PROGRAM prgObjectCode
  VAR
    asPatternName : ARRAY[0..c_uiMaxIndPattern] OF STRING := ['1000L6S4A', '1000L6S5A', '1000L7S2A', '1000L9S0A', '800L2S6A', '800L4S3A', '800L5S2A', '800L6S0A', '800L6S1A'];  (* palletizing options *)
    iTMPMaxIndShowPattern : INT;
    iMaxIndPattern : INT;
    iMaxIndShowPattern : INT;
    iMaxIndLayer : INT;
    iTMPMaxIndShowLayer : INT;
    iMaxIndShowLayer : INT;
    iMaxIndTool : INT;
    iTMPMaxIndShowTool : INT;
    iMaxIndShowTool : INT;
    asToolName : ARRAY[0..c_uiMaxIndTool] OF STRING;
  END_VAR
  VAR CONSTANT
    c_uiMaxIndPattern : UINT := 19;
    c_uiMaxIndTool : UINT := 4;
  END_VAR
  VAR
    asLayerName : ARRAY[0..c_uiMaxIndLayers] OF STRING := ['layer0', 'layer1', 'layer2', 'layer3', 'layer4', 'layer5'];  (* palletizing options *)
  END_VAR
  VAR CONSTANT
    c_uiMaxIndLayers : UINT := 5;
  END_VAR
  VAR
    sDesiredObjectCode01 : STRING;
    sDesiredObjectCode02 : STRING;
    sCurrentObjectCode01 : STRING;
    sCurrentObjectCode02 : STRING;
    xInit : BOOL := TRUE;
    asBoxName : ARRAY[0..c_uiMaxIndBoxTypes] OF STRING := ['SMALL_BOX', 'BIG_BOX'];
    aiDefaultIndex : ARRAY[0..c_uiMaxIndBoxTypes] OF INT := [0, 0];
    iMaxInd : INT;
    iInd : INT;
    iTMPMaxIndShow : INT;
    iMaxIndShow : INT;
  END_VAR
  VAR CONSTANT
    c_uiNumBoxTypes : UINT := 2;
    c_uiMaxIndBoxTypes : UINT := (c_uiNumBoxTypes - 1);
  END_VAR

                    iMaxInd := TO_INT(XSIZEOF(asBoxName)/XSIZEOF(asBoxName[0])) - 1;
(*------------------------------------*)
// find max ind to show
iTMPMaxIndShow := -1;
FOR iInd := 0 TO iMaxInd DO
	IF asBoxName[iInd] <> '' THEN
		iTMPMaxIndShow := iInd;
	END_IF
END_FOR
IF iTMPMaxIndShow >= 0 THEN
	iMaxIndShow := iTMPMaxIndShow;
END_IF
(*------------------------------------*)
// find max ind to show
IF xInit THEN
	xInit := FALSE;
	FOR iInd := 0 TO iMaxInd DO
		CASE iInd OF 
			0:
				METH_SetObjectCode01(sValue := asBoxName[aiDefaultIndex[iInd]]);
			1:
				METH_SetObjectCode02(sValue := asBoxName[aiDefaultIndex[iInd]]);
		END_CASE
	END_FOR
	
END_IF

(*------------------------------------*)
// PATTERN find max ind to show
iMaxIndPattern := TO_INT(XSIZEOF(asPatternName)/XSIZEOF(asPatternName[0])) - 1;
iTMPMaxIndShowPattern := -1;
FOR iInd := 0 TO iMaxIndPattern DO
	IF asPatternName[iInd] <> '' THEN
		iTMPMaxIndShowPattern := iInd;
	END_IF
END_FOR
IF iTMPMaxIndShowPattern >= 0 THEN
	iMaxIndShowPattern := iTMPMaxIndShowPattern;
END_IF
(*------------------------------------*)
// LAYER find max ind to show
iMaxIndLayer := TO_INT(XSIZEOF(asLayerName)/XSIZEOF(asLayerName[0])) - 1;
iTMPMaxIndShowLayer := -1;
FOR iInd := 0 TO iMaxIndLayer DO
	IF asLayerName[iInd] <> '' THEN
		iTMPMaxIndShowLayer := iInd;
	END_IF
END_FOR
IF iTMPMaxIndShowLayer >= 0 THEN
	iMaxIndShowLayer := iTMPMaxIndShowLayer;
END_IF
(*------------------------------------*)
// LAYER find max ind to show
iMaxIndTool := TO_INT(XSIZEOF(asToolName)/XSIZEOF(asToolName[0])) - 1;
iTMPMaxIndShowTool := -1;
FOR iInd := 0 TO iMaxIndTool DO
	IF asToolName[iInd] <> '' THEN
		iTMPMaxIndShowTool := iInd;
	END_IF
END_FOR
IF iTMPMaxIndShowTool >= 0 THEN
	iMaxIndShowTool := iTMPMaxIndShowTool;
END_IF


(*------------------------------------*)
// set ros interface
prgROS.METH_SetObjectName_Left_01(sValue := sCurrentObjectCode01);
prgROS.METH_SetObjectName_Right_01(sValue := sCurrentObjectCode01);
prgROS.METH_SetObjectName_Left_02(sValue := sCurrentObjectCode02);
prgROS.METH_SetObjectName_Right_02(sValue := sCurrentObjectCode02);
// GVL.g_ROSInterface_01.sObjectCode := sCurrentObjectCode01;
// GVL.g_ROSInterface_02.sObjectCode := sCurrentObjectCode02;
                  

METHOD METH_SetObjectCode01
  VAR_INPUT
    sValue : STRING;
  END_VAR
                          sDesiredObjectCode01 := sValue;
METH_SetObjCode01();
                        
END_METHOD

METHOD METH_SetObjectCode02
  VAR_INPUT
    sValue : STRING;
  END_VAR
                          sDesiredObjectCode02 := sValue;
METH_SetObjCode02();

                        
END_METHOD

METHOD METH_SetObjCode02
                          sCurrentObjectCode02 := sDesiredObjectCode02;
                        
END_METHOD

METHOD METH_SetObjCode01
                          sCurrentObjectCode01 := sDesiredObjectCode01;
                        
END_METHOD
END_PROGRAM

PROGRAM prg_Hmi_ObjectCode
  VAR
    xDIS_SetObjCode01 : BOOL;
    xTB_SetObjCode01 : BOOL;
    iIndexObjectCode01 : INT;
    sDesiredObjectCode01 : STRING;
    xDIS_SetObjCode02 : BOOL;
    xTB_SetObjCode02 : BOOL;
    iIndexObjectCode02 : INT;
    sDesiredObjectCode02 : STRING;
    sCurrentObjectCode01 : STRING;
    sCurrentObjectCode02 : STRING;
    sPrevDesiredObjectCode01 : STRING;
    sPrevDesiredObjectCode02 : STRING;
  END_VAR

                    // Object 01
sDesiredObjectCode01 := prgObjectCode.asBoxName[iIndexObjectCode01];
xDIS_SetObjCode01 := sDesiredObjectCode01 = '';
IF sDesiredObjectCode01 <> sPrevDesiredObjectCode01 AND NOT xDIS_SetObjCode01 THEN
	xTB_SetObjCode01 := TRUE;
END_IF
IF xTB_SetObjCode01 THEN
	xTB_SetObjCode01 := FALSE;
	prgObjectCode.METH_SetObjectCode01(sValue := sDesiredObjectCode01);
END_IF
(*------------------------------------*)
// Object 02
sDesiredObjectCode02 := prgObjectCode.asBoxName[iIndexObjectCode02];
xDIS_SetObjCode02 := sDesiredObjectCode02 = '';
IF sDesiredObjectCode02 <> sPrevDesiredObjectCode02 AND NOT xDIS_SetObjCode02 THEN
	xTB_SetObjCode02 := TRUE;
END_IF
IF xTB_SetObjCode02 THEN
	xTB_SetObjCode02 := FALSE;
	prgObjectCode.METH_SetObjectCode02(sValue := sDesiredObjectCode02);
END_IF
(*------------------------------------*)
sCurrentObjectCode01 := prgObjectCode.sCurrentObjectCode01;
sCurrentObjectCode02 := prgObjectCode.sCurrentObjectCode02;


sPrevDesiredObjectCode01 := sDesiredObjectCode01;
sPrevDesiredObjectCode02 := sDesiredObjectCode02;
                  
END_PROGRAM

PROGRAM prgOPCUAIncas
  VAR
    BoxInfo : INCAS_box_info_struct_t;
    sPrevBoxCode : STRING;
    sCurrentBoxCode : STRING;
    xThereIsANewBox : BOOL;
    INCAS_BoxInfo_01 : INCAS_box_info_struct_t;
    INCAS_BoxAck_01 : INCAS_box_ack_struct_t := (time_stamp := 'DT#2023-04-26-17:54:02.008', last_box_code := '123123', error_id := 1);
  END_VAR

                    BoxInfo := INCAS_BoxInfo_01;
(*---------------------------------------*)
sCurrentBoxCode := BoxInfo.box_code;
xThereIsANewBox := sCurrentBoxCode <> sPrevBoxCode AND sCurrentBoxCode <> '';
IF xThereIsANewBox THEN
	prgInboundSync.METH_NewBoxAtGate(BoxInfo := BoxInfo);
END_IF
sPrevBoxCode := BoxInfo.box_code;
                  

METHOD METH_SetIncasInboundFeedback_01 : INT
  VAR_INPUT
    Feedback : INCAS_box_ack_struct_t;
  END_VAR
                          INCAS_BoxAck_01 := Feedback;
                        
END_METHOD
END_PROGRAM

(* {warning 'interrogazione tutte requested action pendenti da fare. Sto facendo'} *)
PROGRAM prgDBQuerier_SorterSX
  VAR
    REQ_CallOutboundProc : SysDesignBasic.FB_SysD_RequestDetail;  (* Call outbound procedure *)
    xTB_CallOutboundProc : BOOL;
    iFailedConsecCallOutboundProc : INT;
    R_TRIG_CallOutboundProcSuccess : R_TRIG;
    R_TRIG_CallOutboundProcFailure : R_TRIG;
    xTB_TESTCallOutboundProc : BOOL;
    iComposeCallProcOutboundRes : INT;
    sOutboundBoxCode : STRING;
    sOutboundGateCode : STRING;
    REQ_CallInboundProc : SysDesignBasic.FB_SysD_RequestDetail;  (* Call inbound procedure *)
    xTB_CallInboundProc : BOOL;
    iFailedConsecCallInboundProc : INT;
    R_TRIG_CallInboundProcSuccess : R_TRIG;
    R_TRIG_CallInboundProcFailure : R_TRIG;
    xTB_TESTCallInboundProc : BOOL;
    iComposeCallProcInboundRes : INT;
    sInboundBoxCode : STRING;
    sInboundGateCode : STRING;
    REQ_GetOutboundCommands : SysDesignBasic.FB_SysD_RequestDetail;  (* GET OUTBOUND COMMANDS *)
    xTB_GetOutboundCommands : BOOL;
    iFailedConsecGetOutboundCommands : INT;
    R_TRIG_GetOutboundCommandsSuccess : R_TRIG;
    R_TRIG_GetOutboundCommandsFailure : R_TRIG;
    xTB_TESTGetOutboundCommands : BOOL;
    aOutboundCommands : ARRAY[0..c_uiOutboundCommandMaxInd] OF db_t_commands_struct_t;
    aOutboundCommandsTMP : ARRAY[0..c_uiOutboundCommandMaxInd] OF db_t_commands_struct_t;
    SQL_Interp_GetOutboundCommands_0 : SQL_Interp_GetCommands;
  END_VAR
  VAR CONSTANT
    c_uiOutboundCommandMaxInd : INT := 9;
  END_VAR
  VAR
    REQ_GetInboundCommands : SysDesignBasic.FB_SysD_RequestDetail;  (* GET INBOUND COMMANDS *)
    xTB_GetInboundCommands : BOOL;
    iFailedConsecGetInboundCommands : INT;
    R_TRIG_GetInboundCommandsSuccess : R_TRIG;
    R_TRIG_GetInboundCommandsFailure : R_TRIG;
    xTB_TESTGetInboundCommands : BOOL;
    aInboundCommands : ARRAY[0..c_uiInboundCommandMaxInd] OF db_t_commands_struct_t;
    aInboundCommandsTMP : ARRAY[0..c_uiInboundCommandMaxInd] OF db_t_commands_struct_t;
    SQL_Interp_GetInboundCommands_0 : SQL_Interp_GetCommands;
  END_VAR
  VAR CONSTANT
    c_uiInboundCommandMaxInd : INT := 9;
  END_VAR
  VAR
    REQ_GetBoxInfo : SysDesignBasic.FB_SysD_RequestDetail;  (* BOX INFO *)
    xTB_GetBoxInfo : BOOL;
    iFailedConsecGetBoxInfo : INT;
    R_TRIG_GetBoxInfoSuccess : R_TRIG;
    R_TRIG_GetBoxInfoFailure : R_TRIG;
    sBoxCode : STRING;
    xTB_TESTGetBoxInfo : BOOL;
    sTESTGetBoxInfo : STRING := 'aaa';
    aBoxInfo : ARRAY[0..c_uiBoxInfoMaxInd] OF db_t_items_struct_t;
    aItemsTMP : ARRAY[0..c_uiBoxInfoMaxInd] OF db_t_items_struct_t;
    SQL_Interp_GetBoxInfo_0 : SQL_Interp_GetItems;
    xTESTIsATest : BOOL := TRUE;
    sINPUTBoxCode : STRING;
    xDEBUG : BOOL := TRUE;
    xShallBeExposed : BOOL;
    xExpose : BOOL;
    iResNotify : INT;
  END_VAR
  VAR CONSTANT
    c_uiBoxInfoNum : UINT := 1;
    c_uiBoxInfoMaxInd : UINT := (c_uiBoxInfoNum - 1);
  END_VAR
  VAR
    xIsSQLQueryAllowed : BOOL;  (* GENERIC QUERYSQL *)
    FB_QuerySQL_0 : SysD_DB.FB_QuerySQL;
    CTRL_Query : SysD_DB.SysD_DB_querier_ctrl_struct_t;
    eMySQLAction : SysD_DB.SysD_DB_actions_enum_t;
    REF_REQ_SQLQuery : REFERENCE TO SysDesignBasic.FB_SysD_RequestDetail;
    REF_REQ_Dummy : SysDesignBasic.FB_SysD_RequestDetail;
    iCountSuccess : INT;  (* counters *)
    iCountFailure : INT;
    eLastQuerierError : SysD_DB.ERROR_QUERIER;  (* errors *)
    eLastInterpError : SysD_DB.ERROR;
    eLastSysD_DB_Error : SysD_DB.ERROR;
    eLastMySQLError : SysD_DB.MySQL.ERROR;
    pDB_INQueue : POINTER TO COL.Queue;  (* pointers to collection elements *)
    pDB_OUTHashTable : POINTER TO COL.IMap;
    SysD_DB_Input : SysD_DB.SysD_db_input_struct_t := (sHost := GVL_Constants.gc_sTESTDatabaseIP, sDatabase := GVL_Constants.gc_sTESTDatabaseName, sUsername := 'plc_user', sPassword := 'deb11_mySQL');  (* database specific *)
    sQuery : SysD_DB.SysD_MySQLQuery;
    iBufferSize : INT;
    xIsValidRef_SQLQueryReq : BOOL;
    asMySQLCommand : SysD_DB.SysD_MySQLCommand;
    diQueryActualLength : DINT;
    pInterpDest : __XWORD;
    uiDimInterpDest : UINT;
    itfInterpreter : SysD_DB.ITF_DBQueryInterpret;
    eErrQuery2Command : SysD_DB.ERROR;
    sAux : STRING(255);
    xNewRowSuccessfullyInserted : BOOL;
  END_VAR
  VAR CONSTANT
    c_sCallerName : STRING := 'PLC';  (* IEC program specific *)
  END_VAR

                    pDB_INQueue := ADR(prgDBExecutor.itfINQueue_MySQLRequest);
pDB_OUTHashTable := ADR(prgDBExecutor.itfOUTHashTable_MySQLResult);

iBufferSize := TO_INT(XSIZEOF(sQuery));

ACT_CheckReferences();
(*====================================================*)
//01/12/2022: set db
// SysD_DB_Input.sHost := GVL.g_sIPCurrentDB; //02/12/2022
// SysD_DB_Input.sDatabase := GVL.g_sNameCurrentDB; //15/03/2023
(*====================================================*)
// // inhibited stations polling
// ACT_InhibitedStationsPolling();
// (*====================================================*)
// // refill stations polling
// ACT_RefillStationsPolling();
// (*====================================================*)
// // output stations polling
// ACT_OutputStationsPolling();
// (*====================================================*)
// // double way stations polling
// ACT_DoubleWayPolling();
// (*====================================================*)
// // current missions polling
// ACT_CurrentMissionsPolling();
// (*====================================================*)
// // delete requested action
// ACT_DeleteRequestedActionTesting();
// (*====================================================*)
// // reschedule requested action
// ACT_RescheduleRequestedActionTesting();
// (*====================================================*)
// // get pending requested action polling
// ACT_GetPendingRequestedActionsPolling();
// (*====================================================*)
// // station enabling
// ACT_StationEnablingTesting();
// (*====================================================*)
// // station two ways
// ACT_StationTwoWaysTesting();
// (*====================================================*)

xIsSQLQueryAllowed := NOT CTRL_Query.xExecute;
IF xIsSQLQueryAllowed THEN
	IF xTB_GetBoxInfo THEN
		xTB_GetBoxInfo := FALSE;
		IF xTESTIsATest THEN
			sBoxCode := sTESTGetBoxInfo;
		ELSE
			sBoxCode := sINPUTBoxCode;
		END_IF
		IF xShallBeExposed THEN
			xShallBeExposed := FALSE;
			xExpose := TRUE;
		END_IF
		ACT_GetBoxInfo_Request();
		REF_REQ_SQLQuery.METH_SetRequested();
		CTRL_Query.xExecute := TRUE;
	ELSIF xTB_GetInboundCommands THEN
		xTB_GetInboundCommands := FALSE;
		ACT_GetInboundCommands_Request();
		REF_REQ_SQLQuery.METH_SetRequested();
		CTRL_Query.xExecute := TRUE;
	ELSIF xTB_GetOutboundCommands THEN
		xTB_GetOutboundCommands := FALSE;
		ACT_GetOutboundCommands_Request();
		REF_REQ_SQLQuery.METH_SetRequested();
		CTRL_Query.xExecute := TRUE;
	END_IF
END_IF
(*---------------------------------------------------------------*)
(*---------------------------------------------------------------*)
// Querier execution
ACT_SQLQuery();
(*---------------------------------------------------------------*)
(*---------------------------------------------------------------*)
// manage results

// 07/02/2023: get BOX INFO from t_item
R_TRIG_GetBoxInfoSuccess(CLK := REQ_GetBoxInfo.METH_IsSuccess());
IF R_TRIG_GetBoxInfoSuccess.Q THEN
	ACT_GetBoxInfo_Success();
END_IF

R_TRIG_GetBoxInfoFailure(CLK := REQ_GetBoxInfo.METH_IsFailure());
IF R_TRIG_GetBoxInfoFailure.Q THEN
	ACT_GetBoxInfo_Failure();
END_IF
(*---------------------------------------------------------------*)
// Get INBOUND COMMANDS
R_TRIG_GetInboundCommandsSuccess(CLK := REQ_GetInboundCommands.METH_IsSuccess());
IF R_TRIG_GetInboundCommandsSuccess.Q THEN
	ACT_GetInboundCommands_Success();
END_IF

R_TRIG_GetInboundCommandsFailure(CLK := REQ_GetInboundCommands.METH_IsFailure());
IF R_TRIG_GetInboundCommandsFailure.Q THEN
	ACT_GetInboundCommands_Failure();
END_IF
(*---------------------------------------------------------------*)
// Get OUTBOUND COMMANDS
R_TRIG_GetOutboundCommandsSuccess(CLK := REQ_GetOutboundCommands.METH_IsSuccess());
IF R_TRIG_GetOutboundCommandsSuccess.Q THEN
	ACT_GetOutboundCommands_Success();
END_IF

R_TRIG_GetOutboundCommandsFailure(CLK := REQ_GetOutboundCommands.METH_IsFailure());
IF R_TRIG_GetOutboundCommandsFailure.Q THEN
	ACT_GetOutboundCommands_Failure();
END_IF
(*---------------------------------------------------------------*)
// Call INBOUND procedure
R_TRIG_GetOutboundCommandsSuccess(CLK := REQ_GetOutboundCommands.METH_IsSuccess());
IF R_TRIG_GetOutboundCommandsSuccess.Q THEN
	ACT_GetOutboundCommands_Success();
END_IF

R_TRIG_GetOutboundCommandsFailure(CLK := REQ_GetOutboundCommands.METH_IsFailure());
IF R_TRIG_GetOutboundCommandsFailure.Q THEN
	ACT_GetOutboundCommands_Failure();
END_IF
(*---------------------------------------------------------------*)

                  

ACTION ACT_GetInhibitedStations_Failure:
                        IF CTRL_Query.xAborted THEN
	//
ELSIF CTRL_Query.xFailure THEN
	//
END_IF

xGettingStationStates := FALSE;
iFailedConsecutively := iFailedConsecutively + 1;

                      
END_ACTION

ACTION ACT_GetInhibitedStations_Success:
                        IF eLastInterpError = SysD_DB.ERROR.NO_ERROR THEN
	diActionID := aStationStatesBuffer[0].diRowNum;
ELSIF eLastInterpError = SysD_DB.ERROR.NULL_RESULT THEN
	diActionID := -1;
END_IF

METH_CopyInhibitedStationBuffer();
xContinueGettingInhibitedStations := METH_IsBufferFull();
IF xContinueGettingInhibitedStations THEN
	xTB_GetInhibitedStations := TRUE;
ELSE
	xGettingStationStates := FALSE;
	aStationStates := aStationStatesTMP;
	diRTCResult := SysTimeRtc.SysTimeRtcHighResGet(pTimestamp := uliLastTimestampInhibitedStations);
END_IF

iFailedConsecutively := 0;
                      
END_ACTION

ACTION ACT_GetInhibitedStations_Request:
                        SysMem.SysMemSet(pDest := ADR(sQuery), udiValue := 0, udiCount := XSIZEOF(sQuery));
SysMem.SysMemSet(pDest := ADR(asMySQLCommand), udiValue := 0, udiCount := XSIZEOF(asMySQLCommand));
iBufferSize := TO_INT(XSIZEOF(sQuery));

ACT_ComposeInhibitedStationsQuery();

diQueryActualLength := STU.StrLenA(pstData := ADR(sQuery));
eErrQuery2Command := SysD_DB.FUN_Query2SQLCmd(
	pbQuery := ADR(sQuery),
	diQueryLength := diQueryActualLength,
	asSQLCommand => asMySQLCommand
);

SysMem.SysMemSet(pDest := ADR(aStationStatesBuffer), udiCount := XSIZEOF(aStationStatesBuffer), udiValue := 0);

pInterpDest := ADR(aStationStatesBuffer);
uiDimInterpDest := __UXINT_TO_UINT(XSIZEOF(aStationStatesBuffer)/XSIZEOF(aStationStatesBuffer[0]));

itfInterpreter := SQL_Interp_GetStationStates_0;

REF_REQ_SQLQuery REF= REQ_GetInhibitedStations;

eMySQLAction := SysD_DB.SysD_DB_actions_enum_t.Query;


                      
END_ACTION

ACTION ACT_ComposeInhibitedStationsQuery:
                        diLastInhibitedStatationsRowNum := METH_GetLastInhibitedStationsID(iIndexFound => iIndexLastInhibitedStation);
sLastInhibitedStationRowNum := TO_STRING(diLastInhibitedStatationsRowNum);
iAvailableSlots := MIN(
		TO_INT(XSIZEOF(aStationStatesTMP)/XSIZEOF(aStationStatesTMP[0])) - MAX(0, iIndexLastInhibitedStation),
		(c_iMaxRowInd + 1) 
);
sAvailableSpots := TO_STRING(iAvailableSlots);

sQuery := 'select * from v_inhibited_stations where row_num > ';	
STU.StrConcatA(pstTo := ADR(sQuery), pstFrom := ADR(sLastInhibitedStationRowNum), iBufferSize := TO_INT(XSIZEOF(sQuery)));
STU.StrConcatA(pstTo := ADR(sQuery), pstFrom := ADR(' limit '), iBufferSize := TO_INT(XSIZEOF(sQuery)));
STU.StrConcatA(pstTo := ADR(sQuery), pstFrom := ADR(sAvailableSpots), iBufferSize := TO_INT(XSIZEOF(sQuery)));
// STU.StrConcatA(pstTo := ADR(sQuery), pstFrom := ADR(';'), iBufferSize := TO_INT(XSIZEOF(sQuery)));
                      
END_ACTION

ACTION ACT_InhibitedStationsPolling:
                        IF xInitInhStatPolling THEN
	xInitInhStatPolling := FALSE;
	tInhibitedStationsPolling := tShortPolling;
END_IF
xPollingAlarm := iFailedConsecutively >= iMaxFailedConsecutively;
TON_PollInhibitedStations(IN := (GVL.g_sIPCurrentDB <> ''), PT := tInhibitedStationsPolling);
IF TON_PollInhibitedStations.Q OR xForceInhibitedUpdate THEN
	xForceInhibitedUpdate := FALSE;
	IF NOT xGettingStationStates AND NOT xPollingAlarm THEN
		TON_PollInhibitedStations(IN := FALSE);
		SysMem.SysMemSet(pDest := ADR(aStationStatesTMP), udiCount := XSIZEOF(aStationStatesTMP), udiValue := 0);
		xTB_GetInhibitedStations := TRUE;
	END_IF
END_IF
                      
END_ACTION

ACTION ACT_GetMissionID_Request:
                        asMySQLCommand[0] := FUN_SAPA_select_mission_id(
	diGMSInstanceID := diGMSInstanceID,
);

pInterpDest := ADR(diAuxMissionID);
uiDimInterpDest := __UXINT_TO_UINT(XSIZEOF(diAuxMissionID)/XSIZEOF(diAuxMissionID));

itfInterpreter := SQL_Interp_GetMissionId_0;

REF_REQ_SQLQuery REF= REQ_GetMissionID;

eMySQLAction := SysD_DB.SysD_DB_actions_enum_t.Query;


                      
END_ACTION

ACTION ACT_GetMissionID_Success:
                        IF eLastInterpError = SysD_DB.ERROR.NO_ERROR THEN
	diMissionID := diAuxMissionID;
ELSIF eLastInterpError = SysD_DB.ERROR.NULL_RESULT THEN
	diMissionID := -1;
END_IF
                      
END_ACTION

ACTION ACT_GetMissionID_Failure:
                        IF CTRL_Query.xAborted THEN
	//
ELSIF CTRL_Query.xFailure THEN
	//
END_IF

                      
END_ACTION

ACTION ACT_SQLQuery:
                        FB_QuerySQL_0(
	xExecute := CTRL_Query.xExecute, //CBML
	xAbort := CTRL_Query.xAbort, //CBML
	
	xBusy => CTRL_Query.xProcessing, //CBML
	
	xDone => CTRL_Query.xSuccess, //CBML
	xError => CTRL_Query.xFailure, //CBML
	xAborted => CTRL_Query.xAborted, //CBML
	
	eErrorID => CTRL_Query.eErrorQuerier, // error
	eInterpError => CTRL_Query.eInterpError, // error
	eSysD_DB_Error => CTRL_Query.eSysD_DB_Error, // error
	eMySQLError => CTRL_Query.eMySQLError, // error
	udiAffetedRows => CTRL_Query.udiAffectedRows, // 28/06/2022: affected rows
	
	sCaller := c_sCallerName, // caller name shoud be unique per IEC program
	
	SysD_DB_Input := SysD_DB_Input, // database parameters
	asMySQLCommand := asMySQLCommand, // specific for what we're looking for
	
	eMySQLAction := eMySQLAction, //28/06/2022: expansion to exec
	pDest := pInterpDest, // specific for what we're looking for
	uiDim := uiDimInterpDest, // specific for what we're looking for
	itfInterpreter := itfInterpreter, // specific for what we're looking for
	
	pDB_INQueue := pDB_INQueue, // queue of sql requests
	pDB_OUTHashTable := pDB_OUTHashTable // hashtable of sql results
);
CTRL_Query.xTerminated := CTRL_Query.xSuccess OR CTRL_Query.xFailure OR CTRL_Query.xAborted;
IF CTRL_Query.xTerminated THEN
	// saving last errors
	eLastQuerierError := CTRL_Query.eErrorQuerier;
	eLastInterpError := CTRL_Query.eInterpError;
	eLastSysD_DB_Error := CTRL_Query.eSysD_DB_Error;
	eLastMySQLError := CTRL_Query.eMySQLError;
	
	// result-specific stuff to always do
	IF CTRL_Query.xSuccess THEN
		iCountSuccess := (iCountSuccess + 1) MOD 16#7FFF;
		REF_REQ_SQLQuery.METH_SetSuccess();
	ELSE
		REF_REQ_SQLQuery.METH_SetFailure();
		iCountFailure := (iCountFailure + 1) MOD 16#7FFF;
		IF CTRL_Query.xAborted THEN
			//
		ELSIF CTRL_Query.xFailure THEN
			//
		END_IF 
	END_IF
	CTRL_Query.xExecute := FALSE;
	FB_QuerySQL_0(xExecute := FALSE);
END_IF

                      
END_ACTION

ACTION ACT_CheckReferences:
                        xIsValidRef_SQLQueryReq := __ISVALIDREF(REF_REQ_SQLQuery);
IF NOT xIsValidRef_SQLQueryReq THEN
	REF_REQ_SQLQuery REF= REF_REQ_Dummy;
END_IF
                      
END_ACTION

ACTION ACT_InsertNewAction_Request:
                        asMySQLCommand[0] := FUN_SAPA_insert_new_action_request(
	sStation := sNewAction_Station,
	eTypeOfRequest := eNewAction_TypeOfRequest,
	sContainerCategory := sContainerCategory,
	xIsAutomatic := xNewAction_IsAutomatic
);

pInterpDest := 0;
uiDimInterpDest := 0;

itfInterpreter := 0;

REF_REQ_SQLQuery REF= REQ_InsertNewActionRequest;

eMySQLAction := SysD_DB.SysD_DB_actions_enum_t.Exec;

xNewRowSuccessfullyInserted := FALSE;
                      
END_ACTION

ACTION ACT_InsertNewAction_Failure:
                        IF CTRL_Query.xAborted THEN
	//
ELSIF CTRL_Query.xFailure THEN
	//
END_IF

                      
END_ACTION

ACTION ACT_InsertNewAction_Success:
                        xNewRowSuccessfullyInserted := FALSE;
IF CTRL_Query.udiAffectedRows > 0 THEN
	xNewRowSuccessfullyInserted := TRUE;
END_IF
                      
END_ACTION

ACTION ACT_GetRequestedActions_Failure:
                        IF CTRL_Query.xAborted THEN
	//
ELSIF CTRL_Query.xFailure THEN
	//
END_IF

                      
END_ACTION

ACTION ACT_GetRequestedActions_Request:
                        CASE eWantedRequestedAction OF
	SAPA_type_of_request_enum_t.NOT_SPECIFIED:
		asMySQLCommand[0] := 'select * from t_requested_actions where issued = 0 order by timestamp asc limit 1';
	SAPA_type_of_request_enum_t.PICK_UP:
		asMySQLCommand[0] := 'select * from t_requested_actions where issued = 0 and type_of_request=$'PICK-UP$' ';
		asMySQLCommand[1] := 'order by timestamp asc limit 1';
	SAPA_type_of_request_enum_t.REFILL:
		asMySQLCommand[0] := 'select * from t_requested_actions where issued = 0 and type_of_request=$'REFILL$' ';
		asMySQLCommand[1] := 'order by timestamp asc limit 1';
END_CASE		


SysMem.SysMemSet(pDest := ADR(aSAPA_RequestedActions), udiCount := XSIZEOF(aSAPA_RequestedActions), udiValue := 0);

pInterpDest := ADR(aSAPA_RequestedActions);
uiDimInterpDest := __UXINT_TO_UINT(XSIZEOF(aSAPA_RequestedActions)/XSIZEOF(aSAPA_RequestedActions[0]));

itfInterpreter := SQL_Interp_GetRequestedActions_0;

REF_REQ_SQLQuery REF= REQ_GetNewActionRequest;

eMySQLAction := SysD_DB.SysD_DB_actions_enum_t.Query;


                      
END_ACTION

ACTION ACT_GetRequestedActions_Success:
                        IF eLastInterpError = SysD_DB.ERROR.NO_ERROR THEN
	diActionID := aSAPA_RequestedActions[0].diID;
ELSIF eLastInterpError = SysD_DB.ERROR.NULL_RESULT THEN
	diActionID := -1;
END_IF
                      
END_ACTION

ACTION ACT_StationContainerType_Failure:
                        IF CTRL_Query.xAborted THEN
	//
ELSIF CTRL_Query.xFailure THEN
	//
END_IF

iFailedConsecStationContainerType := iFailedConsecStationContainerType + 1;

                      
END_ACTION

ACTION ACT_StationContainerType_Success:
                        
iFailedConsecStationContainerType := 0;
                      
END_ACTION

ACTION ACT_StationContainerType_Request:
                        SysMem.SysMemSet(pDest := ADR(sQuery), udiValue := 0, udiCount := XSIZEOF(sQuery));
SysMem.SysMemSet(pDest := ADR(asMySQLCommand), udiValue := 0, udiCount := XSIZEOF(asMySQLCommand));
iBufferSize := TO_INT(XSIZEOF(sQuery));

ACT_ComposeStationContainerType();

diQueryActualLength := STU.StrLenA(pstData := ADR(sQuery));
eErrQuery2Command := SysD_DB.FUN_Query2SQLCmd(
	pbQuery := ADR(sQuery),
	diQueryLength := diQueryActualLength,
	asSQLCommand => asMySQLCommand
);

// SysMem.SysMemSet(pDest := ADR(aSAPA_CurrentMissionsTMP), udiCount := XSIZEOF(aSAPA_CurrentMissionsTMP), udiValue := 0);

pInterpDest := 0;
uiDimInterpDest := 0;

itfInterpreter := 0;

REF_REQ_SQLQuery REF= REQ_StationContainerType;

eMySQLAction := SysD_DB.SysD_DB_actions_enum_t.Exec;


                      
END_ACTION

ACTION ACT_ComposeStationContainerType:
                        sQuery := 'update t_stations set container_category = ';

SysMem.SysMemSet(pDest := ADR(sAux), udiCount := XSIZEOF(sAux), udiValue := 0);
sAux := SysD_DB.FUN_ConvertToSQLQueryString(sString := sContainerTypeToSetOnStation);
STU.StrConcatA(pstTo := ADR(sQuery), pstFrom := ADR(sAux), iBufferSize := TO_INT(XSIZEOF(sQuery)));

STU.StrConcatA(pstTo := ADR(sQuery), pstFrom := ADR(' where station_name = '), iBufferSize := TO_INT(XSIZEOF(sQuery)));

// concat station name
SysMem.SysMemSet(pDest := ADR(sAux), udiCount := XSIZEOF(sAux), udiValue := 0);
sAux := SysD_DB.FUN_ConvertToSQLQueryString(sString := sStationToSetContainerType);
STU.StrConcatA(pstTo := ADR(sQuery), pstFrom := ADR(sAux), iBufferSize := TO_INT(XSIZEOF(sQuery)));
                      
END_ACTION

ACTION ACT_StationContainerTypeTesting:
                        IF xTB_TESTStationContainerType THEN
	xTB_TESTStationContainerType := FALSE;
	METH_SetStationContainerCategory(
		sStationName := sTESTStationToSetContainerType,
		sContainerCategory := sTESTContainerType
	);
	METH_StationContainerCategory();
END_IF
                      
END_ACTION

ACTION ACT_GetRefillStations_Failure:
                        IF CTRL_Query.xAborted THEN
	//
ELSIF CTRL_Query.xFailure THEN
	//
END_IF

iRefillFailedConsec := iRefillFailedConsec + 1;

                      
END_ACTION

ACTION ACT_GetRefillStations_Success:
                        IF eLastInterpError = SysD_DB.ERROR.NO_ERROR THEN
	sRefStat := aSAPA_RefillStations[0].sStationName;
	
	// overwrite global variable for scheduling
	METH_UpdateRefillStationGlobal();
	
	METH_SignalDisabledRefillStationsHMI();
	
ELSIF eLastInterpError = SysD_DB.ERROR.NULL_RESULT THEN
	sRefStat := '';
END_IF

iRefillFailedConsec := 0;
                      
END_ACTION

ACTION ACT_GetRefillStations_Request:
                        SysMem.SysMemSet(pDest := ADR(sQuery), udiValue := 0, udiCount := XSIZEOF(sQuery));
SysMem.SysMemSet(pDest := ADR(asMySQLCommand), udiValue := 0, udiCount := XSIZEOF(asMySQLCommand));
iBufferSize := TO_INT(XSIZEOF(sQuery));

ACT_ComposeRefillStationsQuery();

diQueryActualLength := STU.StrLenA(pstData := ADR(sQuery));
eErrQuery2Command := SysD_DB.FUN_Query2SQLCmd(
	pbQuery := ADR(sQuery),
	diQueryLength := diQueryActualLength,
	asSQLCommand => asMySQLCommand
);

SysMem.SysMemSet(pDest := ADR(aSAPA_RefillStations), udiCount := XSIZEOF(aSAPA_RefillStations), udiValue := 0);

pInterpDest := ADR(aSAPA_RefillStations);
uiDimInterpDest := __UXINT_TO_UINT(XSIZEOF(aSAPA_RefillStations)/XSIZEOF(aSAPA_RefillStations[0]));

itfInterpreter := SQL_Interp_GetRefillStations_0;

REF_REQ_SQLQuery REF= REQ_GetRefillStations;

eMySQLAction := SysD_DB.SysD_DB_actions_enum_t.Query;


                      
END_ACTION

ACTION ACT_ComposeRefillStationsQuery:
                        IF xDebugRefill THEN
	sQuery := 'select * from t_stations limit 8';
ELSE
	IF xRefillStationState THEN
		sQuery := 'select * from v_refill_stations_state order by enabled desc, station_name asc limit 8';
	ELSE
		sQuery := 'select station_name, type_of_station, container_category, enabled from t_stations where type_of_station = $'RV$' order by enabled desc, station_name asc limit 8';
	END_IF
	
	
END_IF

                      
END_ACTION

ACTION ACT_RefillStationsPolling:
                        IF xInitRefStatPolling THEN
	xInitRefStatPolling := FALSE;
	tRefillStationsPolling := tShortPolling;
END_IF
xPollingAlarm := iRefillFailedConsec >= iMaxFailedConsecutively;
TON_PollRefillStations(IN := (GVL.g_sIPCurrentDB <> ''), PT := tRefillStationsPolling);
IF TON_PollRefillStations.Q OR xForceRefillUpdate THEN
	xForceRefillUpdate := FALSE;
	IF NOT xPollingAlarm THEN
		TON_PollRefillStations(IN := FALSE);
		xTB_GetRefillStations := TRUE;
	END_IF
END_IF
                      
END_ACTION

ACTION ACT_GetOutputStations_Failure:
                        IF CTRL_Query.xAborted THEN
	//
ELSIF CTRL_Query.xFailure THEN
	//
END_IF

iOutputFailedConsec := iOutputFailedConsec + 1;

                      
END_ACTION

ACTION ACT_GetOutputStations_Success:
                        IF eLastInterpError = SysD_DB.ERROR.NO_ERROR THEN
	sOutStat := aSAPA_OutputStations[0].sStationName;
	
	// overwrite global variable for scheduling
	METH_UpdateOutputStationGlobal();	
	
	METH_SignalDisabledOutputStationsHMI();
	
ELSIF eLastInterpError = SysD_DB.ERROR.NULL_RESULT THEN
	sOutStat := '';
END_IF

iOutputFailedConsec := 0;
                      
END_ACTION

ACTION ACT_GetOutputStations_Request:
                        SysMem.SysMemSet(pDest := ADR(sQuery), udiValue := 0, udiCount := XSIZEOF(sQuery));
SysMem.SysMemSet(pDest := ADR(asMySQLCommand), udiValue := 0, udiCount := XSIZEOF(asMySQLCommand));
iBufferSize := TO_INT(XSIZEOF(sQuery));

ACT_ComposeOutputStationsQuery();

diQueryActualLength := STU.StrLenA(pstData := ADR(sQuery));
eErrQuery2Command := SysD_DB.FUN_Query2SQLCmd(
	pbQuery := ADR(sQuery),
	diQueryLength := diQueryActualLength,
	asSQLCommand => asMySQLCommand
);

SysMem.SysMemSet(pDest := ADR(aSAPA_OutputStations), udiCount := XSIZEOF(aSAPA_OutputStations), udiValue := 0);

pInterpDest := ADR(aSAPA_OutputStations);
uiDimInterpDest := __UXINT_TO_UINT(XSIZEOF(aSAPA_OutputStations)/XSIZEOF(aSAPA_OutputStations[0]));

itfInterpreter := SQL_Interp_GetOutputStations_0;

REF_REQ_SQLQuery REF= REQ_GetOutputStations;

eMySQLAction := SysD_DB.SysD_DB_actions_enum_t.Query;


                      
END_ACTION

ACTION ACT_ComposeOutputStationsQuery:
                        IF xDebugOutput THEN
	sQuery := 'select * from t_stations limit 8';
ELSE
	IF xOutputStationsState THEN
		sQuery := 'select * FROM v_output_stations_state order by enabled desc, station_name asc limit 8';
	ELSE
		sQuery := 'select station_name, type_of_station, container_category, enabled from t_stations where type_of_station = $'RF$' order by enabled desc, station_name asc limit 8';	
	END_IF
	
END_IF

                      
END_ACTION

ACTION ACT_OutputStationsPolling:
                        IF xInitOutStatPolling THEN
	xInitOutStatPolling := FALSE;
	tOutputStationsPolling := tShortPolling;
END_IF
xPollingAlarm := iOutputFailedConsec >= iMaxFailedConsecutively;
TON_PollOutputStations(IN := (GVL.g_sIPCurrentDB <> ''), PT := tOutputStationsPolling);
IF TON_PollOutputStations.Q OR xForceOutputUpdate THEN
	xForceOutputUpdate := FALSE;
	IF NOT xPollingAlarm THEN
		TON_PollOutputStations(IN := FALSE);
		xTB_GetOutputStations := TRUE;
	END_IF
END_IF
                      
END_ACTION

ACTION ACT_GetDoubleWay_Success:
                        IF eLastInterpError = SysD_DB.ERROR.NO_ERROR THEN
// 	diActionID := aStationStatesBuffer[0].diRowNum;
	sPressID := aSAPA_DoubleWayTMP[0].sPressID;
	aSAPA_DoubleWay := aSAPA_DoubleWayTMP;
ELSIF eLastInterpError = SysD_DB.ERROR.NULL_RESULT THEN
// 	diActionID := -1;
END_IF


iFailedConsecDoubleWay := 0;
                      
END_ACTION

ACTION ACT_GetDoubleWay_Failure:
                        IF CTRL_Query.xAborted THEN
	//
ELSIF CTRL_Query.xFailure THEN
	//
END_IF

iFailedConsecDoubleWay := iFailedConsecDoubleWay + 1;

                      
END_ACTION

ACTION ACT_GetDoubleWay_Request:
                        SysMem.SysMemSet(pDest := ADR(sQuery), udiValue := 0, udiCount := XSIZEOF(sQuery));
SysMem.SysMemSet(pDest := ADR(asMySQLCommand), udiValue := 0, udiCount := XSIZEOF(asMySQLCommand));
iBufferSize := TO_INT(XSIZEOF(sQuery));

ACT_ComposeDoubleWayStationsQuery();

diQueryActualLength := STU.StrLenA(pstData := ADR(sQuery));
eErrQuery2Command := SysD_DB.FUN_Query2SQLCmd(
	pbQuery := ADR(sQuery),
	diQueryLength := diQueryActualLength,
	asSQLCommand => asMySQLCommand
);

SysMem.SysMemSet(pDest := ADR(aSAPA_DoubleWayTMP), udiCount := XSIZEOF(aSAPA_DoubleWayTMP), udiValue := 0);

pInterpDest := ADR(aSAPA_DoubleWayTMP);
uiDimInterpDest := __UXINT_TO_UINT(XSIZEOF(aSAPA_DoubleWayTMP)/XSIZEOF(aSAPA_DoubleWayTMP[0]));

itfInterpreter := SQL_Interp_GetDoubleWay_0;

REF_REQ_SQLQuery REF= REQ_GetDoubleWay;

eMySQLAction := SysD_DB.SysD_DB_actions_enum_t.Query;


                      
END_ACTION

ACTION ACT_ComposeDoubleWayStationsQuery:
                        sQuery := 'select * from t_presses_without_empty_mdr_conveyor limit 40';
                      
END_ACTION

ACTION ACT_DoubleWayPolling:
                        IF xInitDoubleWayPolling THEN
	xInitDoubleWayPolling := FALSE;
	tDoubleWayPolling := tShortPolling;
END_IF
xPollingAlarm := iFailedConsecDoubleWay >= iMaxFailedConsecutively;
TON_PollDoubleWay(IN := (GVL.g_sIPCurrentDB <> ''), PT := tDoubleWayPolling);
IF TON_PollDoubleWay.Q OR xForceDoubleWayUpdate THEN
	xForceDoubleWayUpdate := FALSE;
	IF NOT xPollingAlarm THEN
		TON_PollDoubleWay(IN := FALSE);
		xTB_GetDoubleWayStations := TRUE;
	END_IF
END_IF
                      
END_ACTION

ACTION ACT_GetCurrentMissions_Success:
                        IF eLastInterpError = SysD_DB.ERROR.NO_ERROR THEN
	aSAPA_CurrentMissions := aSAPA_CurrentMissionsTMP;
ELSIF eLastInterpError = SysD_DB.ERROR.NULL_RESULT THEN
// 	diActionID := -1;
	aSAPA_CurrentMissions := aSAPA_CurrentMissionsTMP;
END_IF


iFailedConsecCurrentMissions := 0;
                      
END_ACTION

ACTION ACT_GetCurrentMissions_Failure:
                        IF CTRL_Query.xAborted THEN
	//
ELSIF CTRL_Query.xFailure THEN
	//
END_IF

iFailedConsecCurrentMissions := iFailedConsecCurrentMissions + 1;

                      
END_ACTION

ACTION ACT_GetCurrentMissions_Request:
                        SysMem.SysMemSet(pDest := ADR(sQuery), udiValue := 0, udiCount := XSIZEOF(sQuery));
SysMem.SysMemSet(pDest := ADR(asMySQLCommand), udiValue := 0, udiCount := XSIZEOF(asMySQLCommand));
iBufferSize := TO_INT(XSIZEOF(sQuery));

ACT_ComposeCurrentMissionsQuery();

diQueryActualLength := STU.StrLenA(pstData := ADR(sQuery));
eErrQuery2Command := SysD_DB.FUN_Query2SQLCmd(
	pbQuery := ADR(sQuery),
	diQueryLength := diQueryActualLength,
	asSQLCommand => asMySQLCommand
);

SysMem.SysMemSet(pDest := ADR(aSAPA_CurrentMissionsTMP), udiCount := XSIZEOF(aSAPA_CurrentMissionsTMP), udiValue := 0);

pInterpDest := ADR(aSAPA_CurrentMissionsTMP);
uiDimInterpDest := __UXINT_TO_UINT(XSIZEOF(aSAPA_CurrentMissionsTMP)/XSIZEOF(aSAPA_CurrentMissionsTMP[0]));

itfInterpreter := SQL_Interp_GetCurrentMissions_0;

REF_REQ_SQLQuery REF= REQ_GetCurrentMissions;

eMySQLAction := SysD_DB.SysD_DB_actions_enum_t.Query;


                      
END_ACTION

ACTION ACT_ComposeCurrentMissionsQuery:
                        IF xGetAlsoActionInfo THEN
	sQuery := 'SELECT tm.*, tra.station AS act_station, tra.type_of_request AS act_type, tra.timestamp AS act_timestamp, tra.container_category as act_container_category, tra.assoc_sync as act_assoc_sync from t_missions AS tm JOIN t_requested_actions AS tra ON tra.uuid = tm.requested_action_uuid order by tm.created_at desc limit 10';
ELSE
	sQuery := 'select * from t_missions order by created_at desc limit 10';
END_IF
// SELECT tm.*, tra.station AS act_station, tra.type_of_request AS act_type, tra.timestamp AS act_timestamp
// from t_missions AS tm
// JOIN t_requested_actions AS tra ON tra.uuid = tm.requested_action_uuid
// order by tm.created_at desc limit 10
                      
END_ACTION

ACTION ACT_CurrentMissionsPolling:
                        IF xInitCurrentMissionsPolling THEN
	xInitCurrentMissionsPolling := FALSE;
	tCurrentMissionsPolling := tShortPolling;
END_IF
xPollingAlarm := iFailedConsecCurrentMissions >= iMaxFailedConsecutively;
TON_PollCurrentMissions(IN := (GVL.g_sIPCurrentDB <> ''), PT := tCurrentMissionsPolling);
IF TON_PollCurrentMissions.Q OR xForceCurrentMissionsUpdate THEN
	xForceCurrentMissionsUpdate := FALSE;
	IF NOT xPollingAlarm THEN
		TON_PollCurrentMissions(IN := FALSE);
		xTB_GetCurrentMissions := TRUE;
	END_IF
END_IF
                      
END_ACTION

ACTION ACT_ComposeDeleteRequestedAction:
                        IF xUseDeleteProcedure THEN //22/03/2023: deletes both requests if happened during 1st part of 2 ways combo
	sQuery := 'CALL sp_delete_processing_request(';

	SysMem.SysMemSet(pDest := ADR(sAux), udiCount := XSIZEOF(sAux), udiValue := 0);
	sAux := SysD_DB.FUN_ConvertToSQLQueryString(sString := sRequestedActionToDelete);
	STU.StrConcatA(pstTo := ADR(sQuery), pstFrom := ADR(sAux), iBufferSize := TO_INT(XSIZEOF(sQuery)));
	
	STU.StrConcatA(pstTo := ADR(sQuery), pstFrom := ADR(');'), iBufferSize := TO_INT(XSIZEOF(sQuery)));
ELSE
	sQuery := 'delete from t_requested_actions where uuid = ';

	SysMem.SysMemSet(pDest := ADR(sAux), udiCount := XSIZEOF(sAux), udiValue := 0);
	sAux := SysD_DB.FUN_ConvertToSQLQueryString(sString := sRequestedActionToDelete);
	STU.StrConcatA(pstTo := ADR(sQuery), pstFrom := ADR(sAux), iBufferSize := TO_INT(XSIZEOF(sQuery)));
END_IF


                      
END_ACTION

ACTION ACT_DeleteRequestedAction_Success:
                        
iFailedConsecDeleteReqAct := 0;
METH_ForcePressesStationsUpdate();
METH_ForcePendingRequestsUpdate();
                      
END_ACTION

ACTION ACT_DeleteRequestedAction_Failure:
                        IF CTRL_Query.xAborted THEN
	//
ELSIF CTRL_Query.xFailure THEN
	//
END_IF

iFailedConsecDeleteReqAct := iFailedConsecDeleteReqAct + 1;

                      
END_ACTION

ACTION ACT_DeleteRequestedAction_Request:
                        SysMem.SysMemSet(pDest := ADR(sQuery), udiValue := 0, udiCount := XSIZEOF(sQuery));
SysMem.SysMemSet(pDest := ADR(asMySQLCommand), udiValue := 0, udiCount := XSIZEOF(asMySQLCommand));
iBufferSize := TO_INT(XSIZEOF(sQuery));

ACT_ComposeDeleteRequestedAction();

diQueryActualLength := STU.StrLenA(pstData := ADR(sQuery));
eErrQuery2Command := SysD_DB.FUN_Query2SQLCmd(
	pbQuery := ADR(sQuery),
	diQueryLength := diQueryActualLength,
	asSQLCommand => asMySQLCommand
);

// SysMem.SysMemSet(pDest := ADR(aSAPA_CurrentMissionsTMP), udiCount := XSIZEOF(aSAPA_CurrentMissionsTMP), udiValue := 0);

pInterpDest := 0;
uiDimInterpDest := 0;

itfInterpreter := 0;

REF_REQ_SQLQuery REF= REQ_DeleteRequestedAction;

eMySQLAction := SysD_DB.SysD_DB_actions_enum_t.Exec;


                      
END_ACTION

ACTION ACT_ComposeMasterDeleteRequestedAction:
                        sQuery := 'delete from t_requested_actions where issued = 0 and uuid = ';

SysMem.SysMemSet(pDest := ADR(sAux), udiCount := XSIZEOF(sAux), udiValue := 0);
sAux := SysD_DB.FUN_ConvertToSQLQueryString(sString := sMasterRequestedActionToDelete);
STU.StrConcatA(pstTo := ADR(sQuery), pstFrom := ADR(sAux), iBufferSize := TO_INT(XSIZEOF(sQuery)));
                      
END_ACTION

ACTION ACT_DeleteRequestedActionTesting:
                        IF xTB_TESTDeleteReqAct THEN
	xTB_TESTDeleteReqAct := FALSE;
	METH_SetRequestedActionToDelete(sUUID := sTESTReqActUUID);
	METH_DeleteRequestedAction();
ELSIF xTB_TESTMasterDeleteReqAct THEN
	xTB_TESTMasterDeleteReqAct := FALSE;
	METH_SetMasterRequestedActionToDelete(sUUID := sTESTReqActUUID);
	METH_MasterDeleteRequestedAction();
END_IF
                      
END_ACTION

ACTION ACT_MasterDeleteRequestedAction_Request:
                        SysMem.SysMemSet(pDest := ADR(sQuery), udiValue := 0, udiCount := XSIZEOF(sQuery));
SysMem.SysMemSet(pDest := ADR(asMySQLCommand), udiValue := 0, udiCount := XSIZEOF(asMySQLCommand));
iBufferSize := TO_INT(XSIZEOF(sQuery));

ACT_ComposeMasterDeleteRequestedAction();

diQueryActualLength := STU.StrLenA(pstData := ADR(sQuery));
eErrQuery2Command := SysD_DB.FUN_Query2SQLCmd(
	pbQuery := ADR(sQuery),
	diQueryLength := diQueryActualLength,
	asSQLCommand => asMySQLCommand
);

// SysMem.SysMemSet(pDest := ADR(aSAPA_CurrentMissionsTMP), udiCount := XSIZEOF(aSAPA_CurrentMissionsTMP), udiValue := 0);

pInterpDest := 0;
uiDimInterpDest := 0;

itfInterpreter := 0;

REF_REQ_SQLQuery REF= REQ_DeleteRequestedAction;

eMySQLAction := SysD_DB.SysD_DB_actions_enum_t.Exec;


                      
END_ACTION

ACTION ACT_RescheduleRequestedAction_Failure:
                        IF CTRL_Query.xAborted THEN
	//
ELSIF CTRL_Query.xFailure THEN
	//
END_IF

iFailedConsecReschedReqAct := iFailedConsecReschedReqAct + 1;

                      
END_ACTION

ACTION ACT_RescheduleRequestedAction_Success:
                        
iFailedConsecReschedReqAct := 0;
                      
END_ACTION

ACTION ACT_RescheduleRequestedAction_Request:
                        SysMem.SysMemSet(pDest := ADR(sQuery), udiValue := 0, udiCount := XSIZEOF(sQuery));
SysMem.SysMemSet(pDest := ADR(asMySQLCommand), udiValue := 0, udiCount := XSIZEOF(asMySQLCommand));
iBufferSize := TO_INT(XSIZEOF(sQuery));

ACT_ComposeRescheduleRequestedAction();

diQueryActualLength := STU.StrLenA(pstData := ADR(sQuery));
eErrQuery2Command := SysD_DB.FUN_Query2SQLCmd(
	pbQuery := ADR(sQuery),
	diQueryLength := diQueryActualLength,
	asSQLCommand => asMySQLCommand
);

// SysMem.SysMemSet(pDest := ADR(aSAPA_CurrentMissionsTMP), udiCount := XSIZEOF(aSAPA_CurrentMissionsTMP), udiValue := 0);

pInterpDest := 0;
uiDimInterpDest := 0;

itfInterpreter := 0;

REF_REQ_SQLQuery REF= REQ_RescheduleRequestedAction;

eMySQLAction := SysD_DB.SysD_DB_actions_enum_t.Exec;


                      
END_ACTION

ACTION ACT_ComposeRescheduleRequestedAction:
                        IF sRescheduleMissionsType = 'PICK-UP' THEN
	sQuery := 'update t_requested_actions set issued = 0, issued_by_robot_id=null, issued_gms_instance_id=null where uuid = ';
ELSIF sRescheduleMissionsType = 'REFILL' THEN
	IF sRescheduleActionType = 'REFILL' THEN
		sQuery := 'update t_requested_actions set issued = 0, issued_by_robot_id=null, issued_gms_instance_id=null where uuid = ';
	ELSIF sRescheduleActionType = 'PICK-UP' THEN
		sQuery := 'update t_requested_actions set refilled = 0, refilled_by_robot_id=null, refilled_gms_instance_id=null where uuid = ';
	ELSE
		sQuery := 'update t_requested_actions set issued = 0, issued_by_robot_id=null, issued_gms_instance_id=null, refilled = 0, refilled_by_robot_id=null, refilled_gms_instance_id=null where uuid = ';
	END_IF
ELSE
	sQuery := 'update t_requested_actions set issued = 0, issued_by_robot_id=null, issued_gms_instance_id=null where uuid = ';
END_IF

// concat uuid
SysMem.SysMemSet(pDest := ADR(sAux), udiCount := XSIZEOF(sAux), udiValue := 0);
sAux := SysD_DB.FUN_ConvertToSQLQueryString(sString := sRequestedActionToReschedule);
STU.StrConcatA(pstTo := ADR(sQuery), pstFrom := ADR(sAux), iBufferSize := TO_INT(XSIZEOF(sQuery)));
                      
END_ACTION

ACTION ACT_RescheduleRequestedActionTesting:
                        IF xTB_TESTRescheduleReqAct THEN
	xTB_TESTRescheduleReqAct := FALSE;
	METH_SetRequestedActionToReschedule(
		sUUID := sTESTReschedReqActUUID,
		sMissionType := sTESTReschedReqActMissionType,
		sActionType := sTESTReschedReqActActionType
	);
	METH_RescheduleRequestedAction();
END_IF
                      
END_ACTION

ACTION ACT_PendingRequestedActions_Request:
                        SysMem.SysMemSet(pDest := ADR(sQuery), udiValue := 0, udiCount := XSIZEOF(sQuery));
SysMem.SysMemSet(pDest := ADR(asMySQLCommand), udiValue := 0, udiCount := XSIZEOF(asMySQLCommand));
iBufferSize := TO_INT(XSIZEOF(sQuery));

ACT_ComposePendingRequestedActionsQuery();

diQueryActualLength := STU.StrLenA(pstData := ADR(sQuery));
eErrQuery2Command := SysD_DB.FUN_Query2SQLCmd(
	pbQuery := ADR(sQuery),
	diQueryLength := diQueryActualLength,
	asSQLCommand => asMySQLCommand
);

SysMem.SysMemSet(pDest := ADR(aSAPA_GetPendingRequestedActionsTMP), udiCount := XSIZEOF(aSAPA_GetPendingRequestedActionsTMP), udiValue := 0);

pInterpDest := ADR(aSAPA_GetPendingRequestedActionsTMP);
uiDimInterpDest := __UXINT_TO_UINT(XSIZEOF(aSAPA_GetPendingRequestedActionsTMP)/XSIZEOF(aSAPA_GetPendingRequestedActionsTMP[0]));

itfInterpreter := SQL_Interp_GetPendingRequestedActions_0;

REF_REQ_SQLQuery REF= REQ_GetPendingRequestedActions;

eMySQLAction := SysD_DB.SysD_DB_actions_enum_t.Query;


                      
END_ACTION

ACTION ACT_PendingRequestedActions_Success:
                        IF eLastInterpError = SysD_DB.ERROR.NO_ERROR THEN
	aSAPA_GetPendingRequestedActions := aSAPA_GetPendingRequestedActionsTMP;
ELSIF eLastInterpError = SysD_DB.ERROR.NULL_RESULT THEN
// 	diActionID := -1;
	aSAPA_GetPendingRequestedActions := aSAPA_GetPendingRequestedActionsTMP;
END_IF

iPendingActions := METH_CountPendingActions();

iFailedConsecGetPendRequests := 0;
                      
END_ACTION

ACTION ACT_PendingRequestedActions_Failure:
                        IF CTRL_Query.xAborted THEN
	//
ELSIF CTRL_Query.xFailure THEN
	//
END_IF

iFailedConsecGetPendRequests := iFailedConsecGetPendRequests + 1;

                      
END_ACTION

ACTION ACT_ComposePendingRequestedActionsQuery:
                        sQuery := 'select * from t_requested_actions where (issued = 0 AND type_of_request=$'REFILL$') OR ((issued = 0 and refilled_gms_instance_id IS null) and type_of_request=$'PICK-UP$') limit ';
sAux := TO_STRING(XSIZEOF(aSAPA_GetPendingRequestedActionsTMP)/XSIZEOF(aSAPA_GetPendingRequestedActionsTMP[0]));
STU.StrConcatA(pstTo := ADR(sQuery), pstFrom := ADR(sAux), iBufferSize := TO_INT(XSIZEOF(sQuery)));
                      
END_ACTION

ACTION ACT_GetPendingRequestedActionsPolling:
                        IF xInitPendingRequestedActionsPolling THEN
	xInitPendingRequestedActionsPolling := FALSE;
	tPendingRequestedActionsPolling := tShortPolling;
END_IF
xPollingAlarm := iFailedConsecGetPendRequests >= iMaxFailedConsecutively;
TON_PollPendingRequestedActions(IN := (GVL.g_sIPCurrentDB <> ''), PT := tPendingRequestedActionsPolling);
IF TON_PollPendingRequestedActions.Q OR xForcePendingReqActUpdate THEN
	xForcePendingReqActUpdate := FALSE;
	IF NOT xPollingAlarm THEN
		TON_PollPendingRequestedActions(IN := FALSE);
		xTB_GetPendingRequestedActions := TRUE;
	END_IF
END_IF
                      
END_ACTION

ACTION ACT_StationEnabling_Failure:
                        IF CTRL_Query.xAborted THEN
	//
ELSIF CTRL_Query.xFailure THEN
	//
END_IF

iFailedConsecStationEnabling := iFailedConsecStationEnabling + 1;

                      
END_ACTION

ACTION ACT_StationEnabling_Success:
                        
iFailedConsecStationEnabling := 0;

CASE eStationEnablingType OF
	SAPA_station_types_enum_t.PR:
		METH_ForcePressesStationsUpdate();
	(*---------------------------*)
	SAPA_station_types_enum_t.RF:
		METH_ForceOutputStationsUpdate();
	(*---------------------------*)
	SAPA_station_types_enum_t.RV:
		METH_ForceRefillStationsUpdate();
	(*---------------------------*)
	ELSE
		METH_ForcePressesStationsUpdate();
END_CASE

                      
END_ACTION

ACTION ACT_StationEnabling_Request:
                        SysMem.SysMemSet(pDest := ADR(sQuery), udiValue := 0, udiCount := XSIZEOF(sQuery));
SysMem.SysMemSet(pDest := ADR(asMySQLCommand), udiValue := 0, udiCount := XSIZEOF(asMySQLCommand));
iBufferSize := TO_INT(XSIZEOF(sQuery));

ACT_ComposeStationEnabling();

diQueryActualLength := STU.StrLenA(pstData := ADR(sQuery));
eErrQuery2Command := SysD_DB.FUN_Query2SQLCmd(
	pbQuery := ADR(sQuery),
	diQueryLength := diQueryActualLength,
	asSQLCommand => asMySQLCommand
);

// SysMem.SysMemSet(pDest := ADR(aSAPA_CurrentMissionsTMP), udiCount := XSIZEOF(aSAPA_CurrentMissionsTMP), udiValue := 0);

pInterpDest := 0;
uiDimInterpDest := 0;

itfInterpreter := 0;

REF_REQ_SQLQuery REF= REQ_StationEnabling;

eMySQLAction := SysD_DB.SysD_DB_actions_enum_t.Exec;


                      
END_ACTION

ACTION ACT_ComposeStationEnabling:
                        sQuery := 'update t_stations set enabled = ';
IF xEnableStation THEN
	STU.StrConcatA(pstTo := ADR(sQuery), pstFrom := ADR('1'), iBufferSize := TO_INT(XSIZEOF(sQuery)));
ELSE
	STU.StrConcatA(pstTo := ADR(sQuery), pstFrom := ADR('0'), iBufferSize := TO_INT(XSIZEOF(sQuery)));
END_IF

STU.StrConcatA(pstTo := ADR(sQuery), pstFrom := ADR(' where station_name = '), iBufferSize := TO_INT(XSIZEOF(sQuery)));

// concat station name
SysMem.SysMemSet(pDest := ADR(sAux), udiCount := XSIZEOF(sAux), udiValue := 0);
sAux := SysD_DB.FUN_ConvertToSQLQueryString(sString := sStationToSetEnabling);
STU.StrConcatA(pstTo := ADR(sQuery), pstFrom := ADR(sAux), iBufferSize := TO_INT(XSIZEOF(sQuery)));


eStationEnablingType := SAPA_station_types_enum_t.Unspecified;
IF FIND(sStationToSetEnabling, 'PR') > 0 THEN
	eStationEnablingType := SAPA_station_types_enum_t.PR;
ELSIF FIND(sStationToSetEnabling, 'RF') > 0 THEN
	eStationEnablingType := SAPA_station_types_enum_t.RF;
ELSIF FIND(sStationToSetEnabling, 'RV') > 0 THEN
	eStationEnablingType := SAPA_station_types_enum_t.RV;
END_IF
                      
END_ACTION

ACTION ACT_StationEnablingTesting:
                        IF xTB_TESTStationEnabling THEN
	xTB_TESTStationEnabling := FALSE;
	METH_SetStationEnabling(
		sStationName := sTESTStationToEnable,
		xEnable := xTESTStationEnablingState
	);
	METH_StationEnabling();
END_IF
                      
END_ACTION

ACTION ACT_StationTwoWays_Failure:
                        IF CTRL_Query.xAborted THEN
	//
ELSIF CTRL_Query.xFailure THEN
	//
END_IF

iFailedConsecStationTwoWays := iFailedConsecStationTwoWays + 1;

                      
END_ACTION

ACTION ACT_StationTwoWays_Success:
                        
iFailedConsecStationEnabling := 0;

METH_ForceDoubleWayUpdate();


                      
END_ACTION

ACTION ACT_StationTwoWays_Request:
                        SysMem.SysMemSet(pDest := ADR(sQuery), udiValue := 0, udiCount := XSIZEOF(sQuery));
SysMem.SysMemSet(pDest := ADR(asMySQLCommand), udiValue := 0, udiCount := XSIZEOF(asMySQLCommand));
iBufferSize := TO_INT(XSIZEOF(sQuery));

ACT_ComposeStationTwoWays();

diQueryActualLength := STU.StrLenA(pstData := ADR(sQuery));
eErrQuery2Command := SysD_DB.FUN_Query2SQLCmd(
	pbQuery := ADR(sQuery),
	diQueryLength := diQueryActualLength,
	asSQLCommand => asMySQLCommand
);

// SysMem.SysMemSet(pDest := ADR(aSAPA_CurrentMissionsTMP), udiCount := XSIZEOF(aSAPA_CurrentMissionsTMP), udiValue := 0);

pInterpDest := 0;
uiDimInterpDest := 0;

itfInterpreter := 0;

REF_REQ_SQLQuery REF= REQ_StationTwoWays;

eMySQLAction := SysD_DB.SysD_DB_actions_enum_t.Exec;


                      
END_ACTION

ACTION ACT_ComposeStationTwoWays:
                        IF xIsTwoWays THEN
	sQuery := 'insert into t_presses_without_empty_mdr_conveyor(press_id) values (';
	// concat press base name
	SysMem.SysMemSet(pDest := ADR(sAux), udiCount := XSIZEOF(sAux), udiValue := 0);
	sAux := SysD_DB.FUN_ConvertToSQLQueryString(sString := sStationToSetTwoWays);
	STU.StrConcatA(pstTo := ADR(sQuery), pstFrom := ADR(sAux), iBufferSize := TO_INT(XSIZEOF(sQuery)));
	
	STU.StrConcatA(pstTo := ADR(sQuery), pstFrom := ADR(')'), iBufferSize := TO_INT(XSIZEOF(sQuery)));
ELSE
	sQuery := 'delete from t_presses_without_empty_mdr_conveyor where press_id = ';
	// concat press base name
	SysMem.SysMemSet(pDest := ADR(sAux), udiCount := XSIZEOF(sAux), udiValue := 0);
	sAux := SysD_DB.FUN_ConvertToSQLQueryString(sString := sStationToSetTwoWays);
	STU.StrConcatA(pstTo := ADR(sQuery), pstFrom := ADR(sAux), iBufferSize := TO_INT(XSIZEOF(sQuery)));
END_IF
                      
END_ACTION

ACTION ACT_StationTwoWaysTesting:
                        IF xTB_TESTStationTwoWays THEN
	xTB_TESTStationTwoWays := FALSE;
	METH_SetStationTwoWays(
		sStationName := sTESTStationToTwoWays,
		xTwoWays := xTESTStationIsTwoWays
	);
	METH_StationTwoWays();
END_IF
                      
END_ACTION

ACTION ACT_GetBoxInfo_Success:
                        IF eLastInterpError = SysD_DB.ERROR.NO_ERROR THEN
	aBoxInfo := aItemsTMP;
ELSIF eLastInterpError = SysD_DB.ERROR.NULL_RESULT THEN
// 	diActionID := -1;
	aBoxInfo := aItemsTMP;
END_IF

IF xExpose THEN
	xExpose := FALSE;
	iResNotify := prgInboundSync.METH_NotifyBoxInfo(
		ItemInfo := aBoxInfo[0]
	);
END_IF

iFailedConsecGetBoxInfo := 0;
                      
END_ACTION

ACTION ACT_GetBoxInfo_Failure:
                        IF CTRL_Query.xAborted THEN
	//
ELSIF CTRL_Query.xFailure THEN
	//
END_IF

iFailedConsecGetBoxInfo := iFailedConsecGetBoxInfo + 1;

                      
END_ACTION

ACTION ACT_GetBoxInfo_Request:
                        SysMem.SysMemSet(pDest := ADR(sQuery), udiValue := 0, udiCount := XSIZEOF(sQuery));
SysMem.SysMemSet(pDest := ADR(asMySQLCommand), udiValue := 0, udiCount := XSIZEOF(asMySQLCommand));
iBufferSize := TO_INT(XSIZEOF(sQuery));

IF xDEBUG THEN
	sQuery := 'select * from t_item limit 1';
	sQuery := 'select * from t_item where box_code=$'aaa$' limit 1';
ELSE
	ACT_ComposeGetBoxInfo();
END_IF


diQueryActualLength := STU.StrLenA(pstData := ADR(sQuery));
eErrQuery2Command := SysD_DB.FUN_Query2SQLCmd(
	pbQuery := ADR(sQuery),
	diQueryLength := diQueryActualLength,
	asSQLCommand => asMySQLCommand
);

SysMem.SysMemSet(pDest := ADR(aItemsTMP), udiCount := XSIZEOF(aItemsTMP), udiValue := 0);

pInterpDest := ADR(aItemsTMP);
uiDimInterpDest := __UXINT_TO_UINT(XSIZEOF(aItemsTMP)/XSIZEOF(aItemsTMP[0]));

itfInterpreter := SQL_Interp_GetBoxInfo_0;

REF_REQ_SQLQuery REF= REQ_GetBoxInfo;

eMySQLAction := SysD_DB.SysD_DB_actions_enum_t.Query;


                      
END_ACTION

ACTION ACT_ComposeGetBoxInfo:
                        sQuery := 'select * from t_item where box_code=';
SysMem.SysMemSet(pDest := ADR(sAux), udiCount := XSIZEOF(sAux), udiValue := 0);
sAux := SysD_DB.FUN_ConvertToSQLQueryString(sString := sBoxCode);
STU.StrConcatA(pstTo := ADR(sQuery), pstFrom := ADR(sAux), iBufferSize := iBufferSize);
STU.StrConcatA(pstTo := ADR(sQuery), pstFrom := ADR(' limit 1'), iBufferSize := iBufferSize);
                      
END_ACTION

ACTION ACT_GetInboundCommands_Success:
                        IF eLastInterpError = SysD_DB.ERROR.NO_ERROR THEN
// 	aBoxInfo := aItemsTMP;
ELSIF eLastInterpError = SysD_DB.ERROR.NULL_RESULT THEN
// 	diActionID := -1;
// 	aBoxInfo := aItemsTMP;
END_IF

// IF xExpose THEN
// 	xExpose := FALSE;
// 	iResNotify := prgInboundSync.METH_NotifyBoxInfo(
// 		ItemInfo := aBoxInfo[0]
// 	);
// END_IF

iFailedConsecGetInboundCommands := 0;
                      
END_ACTION

ACTION ACT_GetInboundCommands_Failure:
                        IF CTRL_Query.xAborted THEN
	//
ELSIF CTRL_Query.xFailure THEN
	//
END_IF

iFailedConsecGetInboundCommands := iFailedConsecGetInboundCommands + 1;

                      
END_ACTION

ACTION ACT_GetInboundCommands_Request:
                        SysMem.SysMemSet(pDest := ADR(sQuery), udiValue := 0, udiCount := XSIZEOF(sQuery));
SysMem.SysMemSet(pDest := ADR(asMySQLCommand), udiValue := 0, udiCount := XSIZEOF(asMySQLCommand));
iBufferSize := TO_INT(XSIZEOF(sQuery));

ACT_ComposeGetInboundCommands();

diQueryActualLength := STU.StrLenA(pstData := ADR(sQuery));
eErrQuery2Command := SysD_DB.FUN_Query2SQLCmd(
	pbQuery := ADR(sQuery),
	diQueryLength := diQueryActualLength,
	asSQLCommand => asMySQLCommand
);

SysMem.SysMemSet(pDest := ADR(aInboundCommandsTMP), udiCount := XSIZEOF(aInboundCommandsTMP), udiValue := 0);

pInterpDest := ADR(aInboundCommandsTMP);
uiDimInterpDest := __UXINT_TO_UINT(XSIZEOF(aInboundCommandsTMP)/XSIZEOF(aInboundCommandsTMP[0]));

itfInterpreter := SQL_Interp_GetInboundCommands_0;

REF_REQ_SQLQuery REF= REQ_GetInboundCommands;

eMySQLAction := SysD_DB.SysD_DB_actions_enum_t.Query;


                      
END_ACTION

ACTION ACT_ComposeGetInboundCommands:
                        sQuery := 'select * from t_inbound_command order by id asc';
// SysMem.SysMemSet(pDest := ADR(sAux), udiCount := XSIZEOF(sAux), udiValue := 0);
// sAux := SysD_DB.FUN_ConvertToSQLQueryString(sString := sBoxCode);
// STU.StrConcatA(pstTo := ADR(sQuery), pstFrom := ADR(sAux), iBufferSize := iBufferSize);
// STU.StrConcatA(pstTo := ADR(sQuery), pstFrom := ADR(' limit 1'), iBufferSize := iBufferSize);
                      
END_ACTION

ACTION ACT_GetOutboundCommands_Success:
                        IF eLastInterpError = SysD_DB.ERROR.NO_ERROR THEN
// 	aBoxInfo := aItemsTMP;
ELSIF eLastInterpError = SysD_DB.ERROR.NULL_RESULT THEN
// 	diActionID := -1;
// 	aBoxInfo := aItemsTMP;
END_IF

// IF xExpose THEN
// 	xExpose := FALSE;
// 	iResNotify := prgOutboundSync.METH_NotifyBoxInfo(
// 		ItemInfo := aBoxInfo[0]
// 	);
// END_IF

iFailedConsecGetOutboundCommands := 0;
                      
END_ACTION

ACTION ACT_GetOutboundCommands_Failure:
                        IF CTRL_Query.xAborted THEN
	//
ELSIF CTRL_Query.xFailure THEN
	//
END_IF

iFailedConsecGetOutboundCommands := iFailedConsecGetOutboundCommands + 1;

                      
END_ACTION

ACTION ACT_GetOutboundCommands_Request:
                        SysMem.SysMemSet(pDest := ADR(sQuery), udiValue := 0, udiCount := XSIZEOF(sQuery));
SysMem.SysMemSet(pDest := ADR(asMySQLCommand), udiValue := 0, udiCount := XSIZEOF(asMySQLCommand));
iBufferSize := TO_INT(XSIZEOF(sQuery));

ACT_ComposeGetOutboundCommands();

diQueryActualLength := STU.StrLenA(pstData := ADR(sQuery));
eErrQuery2Command := SysD_DB.FUN_Query2SQLCmd(
	pbQuery := ADR(sQuery),
	diQueryLength := diQueryActualLength,
	asSQLCommand => asMySQLCommand
);

SysMem.SysMemSet(pDest := ADR(aOutboundCommandsTMP), udiCount := XSIZEOF(aOutboundCommandsTMP), udiValue := 0);

pInterpDest := ADR(aOutboundCommandsTMP);
uiDimInterpDest := __UXINT_TO_UINT(XSIZEOF(aOutboundCommandsTMP)/XSIZEOF(aOutboundCommandsTMP[0]));

itfInterpreter := SQL_Interp_GetOutboundCommands_0;

REF_REQ_SQLQuery REF= REQ_GetOutboundCommands;

eMySQLAction := SysD_DB.SysD_DB_actions_enum_t.Query;


                      
END_ACTION

ACTION ACT_ComposeGetOutboundCommands:
                        sQuery := 'select * from t_outbound_command order by id asc';
// SysMem.SysMemSet(pDest := ADR(sAux), udiCount := XSIZEOF(sAux), udiValue := 0);
// sAux := SysD_DB.FUN_ConvertToSQLQueryString(sString := sBoxCode);
// STU.StrConcatA(pstTo := ADR(sQuery), pstFrom := ADR(sAux), iBufferSize := iBufferSize);
// STU.StrConcatA(pstTo := ADR(sQuery), pstFrom := ADR(' limit 1'), iBufferSize := iBufferSize);
                      
END_ACTION

ACTION ACT_CallInboundProc_Request:
                        SysMem.SysMemSet(pDest := ADR(sQuery), udiValue := 0, udiCount := XSIZEOF(sQuery));
SysMem.SysMemSet(pDest := ADR(asMySQLCommand), udiValue := 0, udiCount := XSIZEOF(asMySQLCommand));
iBufferSize := TO_INT(XSIZEOF(sQuery));

ACT_ComposeCallInboundProc();

diQueryActualLength := STU.StrLenA(pstData := ADR(sQuery));
eErrQuery2Command := SysD_DB.FUN_Query2SQLCmd(
	pbQuery := ADR(sQuery),
	diQueryLength := diQueryActualLength,
	asSQLCommand => asMySQLCommand
);

pInterpDest := 0;
uiDimInterpDest := 0;

itfInterpreter := 0;

REF_REQ_SQLQuery REF= REQ_CallInboundProc;

eMySQLAction := SysD_DB.SysD_DB_actions_enum_t.Exec;

xNewRowSuccessfullyInserted := FALSE;
                      
END_ACTION

ACTION ACT_CallInboundProc_Failure:
                        IF CTRL_Query.xAborted THEN
	//
ELSIF CTRL_Query.xFailure THEN
	//
END_IF

iFailedConsecCallInboundProc := iFailedConsecCallInboundProc + 1;

                      
END_ACTION

ACTION ACT_CallInboundProc_Success:
                        xNewRowSuccessfullyInserted := FALSE;
IF CTRL_Query.udiAffectedRows > 0 THEN
	xNewRowSuccessfullyInserted := TRUE;
END_IF

iFailedConsecCallInboundProc := 0;
                      
END_ACTION

ACTION ACT_ComposeCallInboundProc:
                        iComposeCallProcInboundRes := METH_ComposeProcessInboundBox(
	sBoxCode := sInboundBoxCode,
	sGateCode := sInboundGateCode,
	sQueryResult => sQuery,
	diLength => diQueryActualLength
);
                      
END_ACTION

ACTION ACT_CallOutboundProc_Request:
                        SysMem.SysMemSet(pDest := ADR(sQuery), udiValue := 0, udiCount := XSIZEOF(sQuery));
SysMem.SysMemSet(pDest := ADR(asMySQLCommand), udiValue := 0, udiCount := XSIZEOF(asMySQLCommand));
iBufferSize := TO_INT(XSIZEOF(sQuery));

ACT_ComposeCallOutboundProc();

diQueryActualLength := STU.StrLenA(pstData := ADR(sQuery));
eErrQuery2Command := SysD_DB.FUN_Query2SQLCmd(
	pbQuery := ADR(sQuery),
	diQueryLength := diQueryActualLength,
	asSQLCommand => asMySQLCommand
);

pInterpDest := 0;
uiDimInterpDest := 0;

itfInterpreter := 0;

REF_REQ_SQLQuery REF= REQ_CallOutboundProc;

eMySQLAction := SysD_DB.SysD_DB_actions_enum_t.Exec;

xNewRowSuccessfullyInserted := FALSE;
                      
END_ACTION

ACTION ACT_CallOutboundProc_Failure:
                        IF CTRL_Query.xAborted THEN
	//
ELSIF CTRL_Query.xFailure THEN
	//
END_IF

iFailedConsecCallOutboundProc := iFailedConsecCallOutboundProc + 1;

                      
END_ACTION

ACTION ACT_CallOutboundProc_Success:
                        xNewRowSuccessfullyInserted := FALSE;
IF CTRL_Query.udiAffectedRows > 0 THEN
	xNewRowSuccessfullyInserted := TRUE;
END_IF

iFailedConsecCallOutboundProc := 0;
                      
END_ACTION

ACTION ACT_ComposeCallOutboundProc:
                        iComposeCallProcOutboundRes := METH_ComposeProcessOutboundBox(
	sBoxCode := sOutboundBoxCode,
	sQueryResult => sQuery,
	diLength => diQueryActualLength
);
                      
END_ACTION

METHOD METH_GetLastInhibitedStationsID : DINT
  VAR_OUTPUT
    iIndexFound : INT := -1;
  END_VAR
  VAR
    iMaxInd : INT;
    iInd : INT;
    diRes : DINT;
  END_VAR
                          iMaxInd := TO_INT(XSIZEOF(aStationStatesTMP)/XSIZEOF(aStationStatesTMP[0])) - 1;
FOR iInd := 0 TO iMaxInd DO
	IF aStationStatesTMP[iInd].diRowNum > 0 THEN
		diRes := aStationStatesTMP[iInd].diRowNum;
		iIndexFound := iInd;
	ELSE
		EXIT;
	END_IF
END_FOR

METH_GetLastInhibitedStationsID := diRes;
                        
END_METHOD

METHOD METH_IsBufferFull : BOOL
  VAR
    xRes : BOOL;
    iMaxInd : INT;
  END_VAR
                          iMaxInd := TO_INT(XSIZEOF(aStationStatesBuffer)/XSIZEOF(aStationStatesBuffer[0])) - 1;
xRes := aStationStatesBuffer[iMaxInd].diRowNum > 0;

METH_IsBufferFull := xRes;
                        
END_METHOD

METHOD METH_CopyInhibitedStationBuffer
  VAR
    xRes : BOOL;
    iMaxIndBuffer : INT;
    iInd : INT;
    iLastInd : INT;
    iMaxIndDest : INT;
    iTMPInd : INT;
  END_VAR
                          iMaxIndBuffer := TO_INT(XSIZEOF(aStationStatesBuffer)/XSIZEOF(aStationStatesBuffer[0])) - 1;
iMaxIndDest := TO_INT(XSIZEOF(aStationStatesTMP)/XSIZEOF(aStationStatesTMP[0])) - 1;
METH_GetLastInhibitedStationsID(iIndexFound => iLastInd);

iTMPInd := MAX(0, iLastInd);

FOR iInd := 0 TO iMaxIndBuffer DO
	IF iTMPInd + iInd <= iMaxIndDest THEN
		IF aStationStatesBuffer[iInd].diRowNum > 0 THEN
			aStationStatesTMP[iTMPInd + iInd] := aStationStatesBuffer[iInd];
		ELSE 
			EXIT;
		END_IF
	END_IF
END_FOR

                        
END_METHOD

METHOD METH_ClearStationStatesArray : DINT
                          SysMem.SysMemSet(pDest := ADR(aStationStates), udiCount := XSIZEOF(aStationStates), udiValue := 0);
                        
END_METHOD

METHOD METH_UpdateOutputStationGlobal
  VAR
    iInd : INT;
    iMaxInd : INT;
    sStation : STRING;
    iIndLoc : INT;
    iMaxIndLoc : INT;
    iOccupation : INT;
    xIsEnabled : BOOL;
    xBookingBasedOnOccupation : BOOL := TRUE;
  END_VAR
                          // ONLY STATIONS ALREADY EXISTING IN GLOBAL VARIABLE ARE UPDATED!
iMaxInd := TO_INT(XSIZEOF(GVL.g_a_aSAPA_OutputStations[0])/XSIZEOF(GVL.g_a_aSAPA_OutputStations[0][0])) - 1;
iMaxIndLoc := TO_INT(XSIZEOF(aSAPA_OutputStations)/XSIZEOF(aSAPA_OutputStations[0])) - 1;
FOR iInd := 0 TO iMaxInd DO
	sStation := GVL.g_a_aSAPA_OutputStations[0][iInd].sStationName; 
	FOR iIndLoc := 0 TO iMaxIndLoc DO
		IF aSAPA_OutputStations[iIndLoc].sStationName = sStation THEN
			
			iOccupation := aSAPA_OutputStations[iIndLoc].iOccupation; 
			xIsEnabled := aSAPA_OutputStations[iIndLoc].xEnabled;
			
			// copy info from db
			GVL.g_a_aSAPA_OutputStations[0][iInd].xEnabled := xIsEnabled;
// 			GVL.g_a_aSAPA_OutputStations[0][iInd].xBooked := (
// 				aSAPA_OutputStations[iIndLoc].sContainerCategory <> '' 
// 				AND aSAPA_OutputStations[iIndLoc].sContainerCategory <> 'NULL'
// 			);
			GVL.g_a_aSAPA_OutputStations[0][iInd].iOccupation := iOccupation;
			IF xIsEnabled THEN
				CASE iOccupation OF
					0:
						prg_Hmi_Synoptic.METH_SetRFStationAsked(sStation := sStation);
					1:
						prg_Hmi_Synoptic.METH_SetRFStationBeingServed(sStation := sStation);
					ELSE
						prg_Hmi_Synoptic.METH_ResetRFStationError(sStation := sStation);
				END_CASE
			ELSE
				prg_Hmi_Synoptic.METH_SetRFStationDisabled(sStation := sStation);
			END_IF
			
			IF xBookingBasedOnOccupation THEN
				GVL.g_a_aSAPA_OutputStations[0][iInd].xBooked := iOccupation >= 0;
			ELSE
				GVL.g_a_aSAPA_OutputStations[0][iInd].xBooked := (
					aSAPA_OutputStations[iIndLoc].sContainerCategory <> '' 
					AND aSAPA_OutputStations[iIndLoc].sContainerCategory <> 'NULL'
				);
			END_IF
			
			EXIT;
		END_IF
	END_FOR
END_FOR





                        
END_METHOD

METHOD METH_UpdateRefillStationGlobal
  VAR
    iInd : INT;
    iMaxInd : INT;
    sStation : STRING;
    iIndLoc : INT;
    iMaxIndLoc : INT;
    xIsEnabled : BOOL;
    sContCat : SysD_Geek.SysD_Geek_container_category_t;
    iOccupation : INT;
  END_VAR
                          // ONLY STATIONS ALREADY EXISTING IN GLOBAL VARIABLE ARE UPDATED!
iMaxInd := TO_INT(XSIZEOF(PersistentVars.g_a_aSAPA_RefillStations[0])/XSIZEOF(PersistentVars.g_a_aSAPA_RefillStations[0][0])) - 1;
iMaxIndLoc := TO_INT(XSIZEOF(aSAPA_RefillStations)/XSIZEOF(aSAPA_RefillStations[0])) - 1;
FOR iInd := 0 TO iMaxInd DO
	sStation := PersistentVars.g_a_aSAPA_RefillStations[0][iInd].sStationName; 
	FOR iIndLoc := 0 TO iMaxIndLoc DO
		IF aSAPA_RefillStations[iIndLoc].sStationName = sStation THEN
			// copy info from db
			xIsEnabled := aSAPA_RefillStations[iIndLoc].xEnabled;
			sContCat := aSAPA_RefillStations[iIndLoc].sContainerCategory;
			iOccupation := aSAPA_RefillStations[iIndLoc].iOccupation;
			
			IF xIsEnabled THEN
				CASE iOccupation OF
					0:
						prg_Hmi_Synoptic.METH_SetRVStationAsked(sStation := sStation);
					1:
						prg_Hmi_Synoptic.METH_SetRVStationBeingServed(sStation := sStation);			
					ELSE
						prg_Hmi_Synoptic.METH_ResetRVStationError(sStation := sStation);
				END_CASE
			ELSE
				prg_Hmi_Synoptic.METH_SetRVStationDisabled(sStation := sStation);
			END_IF
			
			PersistentVars.g_a_aSAPA_RefillStations[0][iInd].xEnabled := xIsEnabled;
			PersistentVars.g_a_aSAPA_RefillStations[0][iInd].sContainerCategory := sContCat;
			PersistentVars.g_a_aSAPA_RefillStations[0][iInd].iOccupation := iOccupation;
			EXIT;
		END_IF
	END_FOR
END_FOR





                        
END_METHOD

METHOD METH_SignalDisabledRefillStationsHMI
  VAR
    iMaxInd : INT;
    iInd : INT;
    sStation : STRING;
  END_VAR
                          iMaxInd := TO_INT(XSIZEOF(PersistentVars.g_a_aSAPA_RefillStations[0])/XSIZEOF(PersistentVars.g_a_aSAPA_RefillStations[0][0])) - 1;
FOR iInd := 0 TO iMaxInd DO
	sStation := PersistentVars.g_a_aSAPA_RefillStations[0][iInd].sStationName; 
	IF PersistentVars.g_a_aSAPA_RefillStations[0][iInd].xEnabled THEN
		prg_Hmi_Synoptic.METH_SetRVStationEnable(sStation := sStation);
	ELSE	
		prg_Hmi_Synoptic.METH_SetRVStationDisabled(sStation := sStation);
	END_IF
END_FOR
                        
END_METHOD

METHOD METH_SignalDisabledOutputStationsHMI
  VAR
    iMaxInd : INT;
    iInd : INT;
    sStation : STRING;
  END_VAR
                          iMaxInd := TO_INT(XSIZEOF(GVL.g_a_aSAPA_OutputStations[0])/XSIZEOF(GVL.g_a_aSAPA_OutputStations[0][0])) - 1;
FOR iInd := 0 TO iMaxInd DO
	sStation := GVL.g_a_aSAPA_OutputStations[0][iInd].sStationName; 
	IF GVL.g_a_aSAPA_OutputStations[0][iInd].xEnabled THEN
		prg_Hmi_Synoptic.METH_SetRFStationEnable(sStation := sStation);
	ELSE
		prg_Hmi_Synoptic.METH_SetRFStationDisabled(sStation := sStation);
	END_IF
END_FOR
                        
END_METHOD

METHOD METH_GotDoubleWayStationsFromDB : BOOL
                          METH_GotDoubleWayStationsFromDB := aSAPA_DoubleWay[0].sPressID <> '';
                        
END_METHOD

METHOD METH_CountPendingActions : INT
  VAR
    iMaxInd : INT;
    iInd : INT;
    iRes : INT;
  END_VAR
                          iMaxInd := TO_INT(XSIZEOF(aSAPA_GetPendingRequestedActions)/XSIZEOF(aSAPA_GetPendingRequestedActions[0])) - 1;

FOR iInd := 0 TO iMaxInd DO
	IF aSAPA_GetPendingRequestedActions[iInd].diID <> 0 THEN
		iRes := iRes + 1;
	ELSE
		EXIT;
	END_IF
END_FOR

METH_CountPendingActions := iRes;
                        
END_METHOD

METHOD METH_CopyInhibitedStationStates
  VAR_OUTPUT
    aInhibitedStations : ARRAY[0..GVL_Constants.gc_iMaxIndStationStates] OF station_problems_struct_t;
  END_VAR
  VAR
    uliLastTimestampInhibitedStations : ULINT;
    aRes : ARRAY[0..GVL_Constants.gc_iMaxIndStationStates] OF station_problems_struct_t;
  END_VAR
                          aRes := aStationStates;
aInhibitedStations := aRes;
                        
END_METHOD

METHOD METH_IsThereAnUpdate : BOOL
  VAR_INPUT
    uliLastUpdatedAt : ULINT;
  END_VAR
                          METH_IsThereAnUpdate := uliLastUpdatedAt < uliLastTimestampInhibitedStations;
                        
END_METHOD

METHOD METH_ForceOutputStationsUpdate
                          xForceOutputUpdate := TRUE;
                        
END_METHOD

METHOD METH_UpdateAllNow
                          xForceDoubleWayUpdate := TRUE;
xForceOutputUpdate := TRUE;
xForceRefillUpdate := TRUE;
xForceInhibitedUpdate := TRUE;
xForceCurrentMissionsUpdate := TRUE;
                        
END_METHOD

METHOD METH_ForcePressesStationsUpdate
                          xForceInhibitedUpdate := TRUE;
                        
END_METHOD

METHOD METH_ForceCurrentMissionsUpdate
                          xForceCurrentMissionsUpdate := TRUE;
                        
END_METHOD

METHOD METH_ForcePendingRequestsUpdate
                          xForcePendingReqActUpdate := TRUE;
                        
END_METHOD

METHOD METH_ForceRefillStationsUpdate
                          xForceRefillUpdate := TRUE;
                        
END_METHOD

METHOD METH_ForceDoubleWayUpdate
                          xForceDoubleWayUpdate := TRUE;
                        
END_METHOD

METHOD METH_GetDoubleWayPressRefill : BOOL
  VAR_INPUT
    sStationCode : SysD_Geek.SysD_Geek_station_t;
    xInfoOnDB : BOOL := TRUE;
  END_VAR
  VAR
    iInd : INT;
    iMaxInd : INT;
    sToFind : STRING;
    xRes : BOOL;
    xGotInfoFromDB : BOOL;
    xOnDB : BOOL;
  END_VAR
                          xGotInfoFromDB := METH_GotDoubleWayStationsFromDB();
xOnDB := xInfoOnDB AND xGotInfoFromDB;
iMaxInd := TO_INT(XSIZEOF(aSAPA_DoubleWay)/XSIZEOF(aSAPA_DoubleWay[0])) - 1;

IF xOnDB THEN
	FOR iInd := 0 TO iMaxInd DO
		sToFind := aSAPA_DoubleWay[iInd].sPressID;
		IF sToFind <> '' THEN
			xRes := FIND(sStationCode, sToFind) > 0;
			IF xRes THEN
				EXIT;
			END_IF
		ELSE
			EXIT;
		END_IF
	END_FOR
ELSE // hard coded
	xRes := 
		FIND(sStationCode, 'PR17') > 0
		OR FIND(sStationCode, 'PR18') > 0
		OR FIND(sStationCode, 'PR19') > 0
		OR FIND(sStationCode, 'PR20') > 0
		OR FIND(sStationCode, 'PR21') > 0
		OR FIND(sStationCode, 'PR22') > 0
		OR FIND(sStationCode, 'PR23') > 0
		OR FIND(sStationCode, 'PR24') > 0
		OR FIND(sStationCode, 'PR25') > 0
		OR FIND(sStationCode, 'PR26') > 0
		OR FIND(sStationCode, 'PR27') > 0
		OR FIND(sStationCode, 'PR31') > 0
	;
END_IF

METH_GetDoubleWayPressRefill := xRes;
	
                        
END_METHOD

METHOD METH_GetDoubleWayPressRefillNum : BOOL
  VAR_INPUT
    sStationNum : STRING;
    xInfoOnDB : BOOL := TRUE;
  END_VAR
  VAR
    iInd : INT;
    iMaxInd : INT;
    sToFind : STRING;
    xRes : BOOL;
    xGotInfoFromDB : BOOL;
    xOnDB : BOOL;
  END_VAR
                          xGotInfoFromDB := METH_GotDoubleWayStationsFromDB();
xOnDB := xInfoOnDB AND xGotInfoFromDB;
iMaxInd := TO_INT(XSIZEOF(aSAPA_DoubleWay)/XSIZEOF(aSAPA_DoubleWay[0])) - 1;

IF xOnDB THEN
	FOR iInd := 0 TO iMaxInd DO
		sToFind := RIGHT(aSAPA_DoubleWay[iInd].sPressID, 2);
		IF sToFind <> '' THEN
			xRes := FIND(sStationNum, sToFind) > 0;
			IF xRes THEN
				EXIT;
			END_IF
		ELSE
			EXIT;
		END_IF
	END_FOR
ELSE // hard coded
	xRes := 
		FIND(sStationNum, '17') > 0
		OR FIND(sStationNum, '18') > 0
		OR FIND(sStationNum, '19') > 0
		OR FIND(sStationNum, '20') > 0
		OR FIND(sStationNum, '21') > 0
		OR FIND(sStationNum, '22') > 0
		OR FIND(sStationNum, '23') > 0
		OR FIND(sStationNum, '24') > 0
		OR FIND(sStationNum, '25') > 0
		OR FIND(sStationNum, '26') > 0
		OR FIND(sStationNum, '27') > 0
		OR FIND(sStationNum, '31') > 0
	;
END_IF

METH_GetDoubleWayPressRefillNum := xRes;
                        
END_METHOD

METHOD METH_IsCodeInRVSet : BOOL
  VAR_INPUT
    sContainerCategory : STRING;
  END_VAR
  VAR
    iMaxInd : INT;
    iInd : INT;
    xRes : BOOL;
  END_VAR
                          iMaxInd := TO_INT(XSIZEOF(PersistentVars.g_a_aSAPA_RefillStations[0])/XSIZEOF(PersistentVars.g_a_aSAPA_RefillStations[0][0])) - 1;
FOR iInd := 0 TO iMaxInd DO
	IF PersistentVars.g_a_aSAPA_RefillStations[0][iInd].sContainerCategory = sContainerCategory THEN
		xRes := PersistentVars.g_a_aSAPA_RefillStations[0][iInd].xEnabled;
		IF xRes THEN
			EXIT;
		END_IF
	END_IF
END_FOR

METH_IsCodeInRVSet := xRes;
                        
END_METHOD

METHOD METH_GetCurrentMissionOnAMR : BOOL
  VAR_INPUT
    sRobotID : STRING;
    diInstanceID : DINT := 0;  (* backup criteria *)
  END_VAR
  VAR_OUTPUT
    CurrentMission : SAPA_missions_struct_t;
  END_VAR
  VAR CONSTANT
    c_NoMission : SAPA_missions_struct_t := (diGMSInstance := 0, sFromStation := '', sToStation := '');
  END_VAR
  VAR
    iInd : INT;
    iMaxInd : INT;
    xMatchingRobot : BOOL;
    xMatchingInstanceID : BOOL;
    xMatchingCriteria : BOOL;
    xRes : BOOL;
  END_VAR
                          iMaxInd := TO_INT(XSIZEOF(aSAPA_CurrentMissions)/XSIZEOF(aSAPA_CurrentMissions[0])) - 1;
FOR iInd := 0 TO iMaxInd DO
	xMatchingRobot := sRobotID = aSAPA_CurrentMissions[iInd].sRobotID;
	xMatchingInstanceID := diInstanceID <> 0 AND diInstanceID = aSAPA_CurrentMissions[iInd].diGMSInstance;
	xMatchingCriteria := xMatchingRobot OR xMatchingInstanceID;
	IF xMatchingCriteria THEN
		xRes := TRUE;
		CurrentMission := aSAPA_CurrentMissions[iInd];
		EXIT;
	ELSE
		CurrentMission := c_NoMission;
	END_IF
END_FOR

METH_GetCurrentMissionOnAMR := xRes;
                        
END_METHOD

METHOD METH_DeleteRequestedAction
                          xTB_DeleteRequestedAction := TRUE;
                        
END_METHOD

METHOD METH_SetMasterRequestedActionToDelete
  VAR_INPUT
    sUUID : STRING;
  END_VAR
                          sMasterRequestedActionToDelete := sUUID;

                        
END_METHOD

METHOD METH_SetRequestedActionToDelete
  VAR_INPUT
    sUUID : STRING;
  END_VAR
                          sRequestedActionToDelete := sUUID;

                        
END_METHOD

METHOD METH_MasterDeleteRequestedAction
                          xTB_MasterDeleteRequestedAction := TRUE;
                        
END_METHOD

METHOD METH_ClearRequestedActionToDelete
                          METH_SetRequestedActionToDelete(sUUID := '');

                        
END_METHOD

METHOD METH_RescheduleRequestedAction
                          xTB_RescheduleRequestedAction := TRUE;
                        
END_METHOD

METHOD METH_SetRequestedActionToReschedule
  VAR_INPUT
    sUUID : STRING;
    sMissionType : STRING;
    sActionType : STRING;
  END_VAR
                          sRequestedActionToReschedule := sUUID;
sRescheduleMissionsType := sMissionType;
sActionType := sActionType;

                        
END_METHOD

METHOD METH_ClearRequestedActionToReschedule
                          METH_SetRequestedActionToReschedule(sUUID := '', sActionType := '', sMissionType := '');

                        
END_METHOD

METHOD METH_GetPendingActionsByPress : INT
  VAR_INPUT
    sPress : STRING;
  END_VAR
  VAR_OUTPUT
    aPendingActionsPress : ARRAY[0..2] OF SAPA_requested_actions_struct_t;
  END_VAR
  VAR
    iRes : INT;  (* aRes : ARRAY[0..2] OF SAPA_requested_actions_struct_t; *)
    iMaxInd : INT;
    iInd : INT;
    xIsPressRelated : BOOL;
    sStation : STRING;
    xIsSX : BOOL;
    xIsDX : BOOL;
    xIsV : BOOL;
    xDetected : BOOL;
    PendingRequest : SAPA_requested_actions_struct_t;
  END_VAR
                          iMaxInd := TO_INT(XSIZEOF(aSAPA_GetPendingRequestedActions)/XSIZEOF(aSAPA_GetPendingRequestedActions[0])) - 1;

FOR iInd := 0 TO iMaxInd DO
	IF aSAPA_GetPendingRequestedActions[iInd].diID <> 0 THEN
		PendingRequest := aSAPA_GetPendingRequestedActions[iInd];
		sStation := PendingRequest.sStation;
		xIsPressRelated := FIND(sStation, sPress) > 0;
		IF xIsPressRelated THEN
			
			xIsSX := RIGHT(sStation, 1) = 'S';
			xIsDX := RIGHT(sStation, 1) = 'D';
			xIsV := RIGHT(sStation, 1) = 'V';
			xDetected := xIsSX OR xIsDX OR xIsV;
			IF xDetected THEN
				iRes := iRes + 1;
				IF xIsSX THEN
					aPendingActionsPress[GVL_Constants.gc_iIndPressSX] := PendingRequest;
				ELSIF xIsDX THEN
					aPendingActionsPress[GVL_Constants.gc_iIndPressDX] := PendingRequest;
				ELSIF xIsV THEN
					aPendingActionsPress[GVL_Constants.gc_iIndPressV] := PendingRequest;
				END_IF
			END_IF
		END_IF
	ELSE
		EXIT;
	END_IF
END_FOR

METH_GetPendingActionsByPress := iRes;
                        
END_METHOD

METHOD METH_SetStationEnabling
  VAR_INPUT
    sStationName : STRING;
    xEnable : BOOL;
  END_VAR
                          sStationToSetEnabling := sStationName;
xEnableStation := xEnable;
                        
END_METHOD

METHOD METH_StationEnabling
                          xTB_StationEnabling := TRUE;
                        
END_METHOD

METHOD METH_IsStationEnabling : BOOL
                          METH_IsStationEnabling := REQ_StationEnabling.METH_IsRequested() OR REQ_StationEnabling.METH_IsProcessing();
                        
END_METHOD

METHOD METH_SetStationContainerCategory
  VAR_INPUT
    sStationName : STRING;
    sContainerCategory : STRING;
  END_VAR
                          sStationToSetContainerType := sStationName;
sContainerTypeToSetOnStation := sContainerCategory;
                        
END_METHOD

METHOD METH_StationContainerCategory
                          xTB_StationContainerType := TRUE;
                        
END_METHOD

METHOD METH_IsStationContainerCategory : BOOL
                          METH_IsStationContainerCategory := REQ_StationContainerType.METH_IsRequested() OR REQ_StationContainerType.METH_IsProcessing();
                        
END_METHOD

METHOD METH_IsStationTwoWays : BOOL
                          METH_IsStationTwoWays := REQ_StationTwoWays.METH_IsRequested() OR REQ_StationTwoWays.METH_IsProcessing();
                        
END_METHOD

METHOD METH_SetStationTwoWays
  VAR_INPUT
    sStationName : STRING;
    xTwoWays : BOOL;
  END_VAR
                          sStationToSetTwoWays := sStationName;
xIsTwoWays := xTwoWays;
                        
END_METHOD

METHOD METH_StationTwoWays
                          xTB_StationTwoWays := TRUE;
                        
END_METHOD

METHOD METH_FindIfSyncd : BOOL
  VAR_INPUT
    diInstanceID : DINT;
  END_VAR
  VAR_OUTPUT
    xError : BOOL;
  END_VAR
  VAR
    iInd : INT;
    iMaxInd : INT;
    xRes : BOOL;
    xFound : BOOL;
  END_VAR
                          iMaxInd := TO_INT(XSIZEOF(aSAPA_CurrentMissions)/XSIZEOF(aSAPA_CurrentMissions[0])) - 1;
FOR iInd := 0 TO iMaxInd DO
	IF aSAPA_CurrentMissions[iInd].diGMSInstance = diInstanceID THEN
		xFound := TRUE;
		xRes := (
			aSAPA_CurrentMissions[iInd].sActionAssocSync <> ''
			AND FIND(aSAPA_CurrentMissions[iInd].sActionAssocSync, 'NULL') = 0
		);
		EXIT;
	END_IF
END_FOR

xError := NOT xError;
METH_FindIfSyncd := xRes;

                        
END_METHOD

METHOD METH_GetBoxInfo : INT
  VAR_INPUT
    sBoxCode : STRING;
  END_VAR
                          xTB_GetBoxInfo := TRUE;
sINPUTBoxCode := sBoxCode;
xShallBeExposed := TRUE;
                        
END_METHOD

METHOD METH_ComposeProcessInboundBox : INT
  VAR_INPUT
    sBoxCode : STRING;
    sGateCode : STRING;
  END_VAR
  VAR_OUTPUT
    sQueryResult : SysD_DB.SysD_MySQLQuery;
    diLength : DINT;
  END_VAR
  VAR
    sRes : SysD_DB.SysD_MySQLQuery;
    sAux : STRING(255);
    iRes : INT;
  END_VAR
  VAR CONSTANT
    c_sProcName : STRING := 'sp_process_inbound_box';
  END_VAR
                          iBufferSize := TO_INT(XSIZEOF(sRes));

STU.StrConcatA(pstTo := ADR(sRes), pstFrom := ADR('call '), iBufferSize := iBufferSize);
STU.StrConcatA(pstTo := ADR(sRes), pstFrom := ADR(c_sProcName), iBufferSize := iBufferSize);
STU.StrConcatA(pstTo := ADR(sRes), pstFrom := ADR('('), iBufferSize := iBufferSize);
(*---------------------------*)
// BOX CODE
SysMem.SysMemSet(pDest := ADR(sAux), udiCount := XSIZEOF(sAux), udiValue := 0);
sAux := SysD_DB.FUN_ConvertToSQLQueryString(sString := sBoxCode);
STU.StrConcatA(pstTo := ADR(sRes), pstFrom := ADR(sAux), iBufferSize := iBufferSize);
(*---------------------------*)
STU.StrConcatA(pstTo := ADR(sRes), pstFrom := ADR(','), iBufferSize := iBufferSize); // separator
(*---------------------------*)
// GATE CODE
SysMem.SysMemSet(pDest := ADR(sAux), udiCount := XSIZEOF(sAux), udiValue := 0);
sAux := SysD_DB.FUN_ConvertToSQLQueryString(sString := sGateCode);
STU.StrConcatA(pstTo := ADR(sRes), pstFrom := ADR(sAux), iBufferSize := iBufferSize);
(*---------------------------*)
STU.StrConcatA(pstTo := ADR(sRes), pstFrom := ADR(')'), iBufferSize := iBufferSize); // terminator
(*---------------------------*)
diLength := STU.StrLenA(pstData := ADR(sRes));
(*---------------------------*)
sQueryResult := sRes; // OUTPUT

METH_ComposeProcessInboundBox := iRes;
                        
END_METHOD

METHOD METH_ComposeProcessOutboundBox : INT
  VAR_INPUT
    sBoxCode : STRING;
  END_VAR
  VAR_OUTPUT
    sQueryResult : SysD_DB.SysD_MySQLQuery;
    diLength : DINT;
  END_VAR
  VAR
    sRes : SysD_DB.SysD_MySQLQuery;
    sAux : STRING(255);
    iRes : INT;
  END_VAR
  VAR CONSTANT
    c_sProcName : STRING := 'sp_process_outbound_box';
  END_VAR
                          iBufferSize := TO_INT(XSIZEOF(sRes));

STU.StrConcatA(pstTo := ADR(sRes), pstFrom := ADR('call '), iBufferSize := iBufferSize);
STU.StrConcatA(pstTo := ADR(sRes), pstFrom := ADR(c_sProcName), iBufferSize := iBufferSize);
STU.StrConcatA(pstTo := ADR(sRes), pstFrom := ADR('('), iBufferSize := iBufferSize);
(*---------------------------*)
// BOX CODE
SysMem.SysMemSet(pDest := ADR(sAux), udiCount := XSIZEOF(sAux), udiValue := 0);
sAux := SysD_DB.FUN_ConvertToSQLQueryString(sString := sBoxCode);
STU.StrConcatA(pstTo := ADR(sRes), pstFrom := ADR(sAux), iBufferSize := iBufferSize);
(*---------------------------*)
// STU.StrConcatA(pstTo := ADR(sRes), pstFrom := ADR(','), iBufferSize := iBufferSize); // separator
// (*---------------------------*)
// // GATE CODE
// SysMem.SysMemSet(pDest := ADR(sAux), udiCount := XSIZEOF(sAux), udiValue := 0);
// sAux := SysD_DB.FUN_ConvertToSQLQueryString(sString := sGateCode);
// STU.StrConcatA(pstTo := ADR(sRes), pstFrom := ADR(sAux), iBufferSize := iBufferSize);
(*---------------------------*)
STU.StrConcatA(pstTo := ADR(sRes), pstFrom := ADR(')'), iBufferSize := iBufferSize); // terminator
(*---------------------------*)
diLength := STU.StrLenA(pstData := ADR(sRes));
(*---------------------------*)
sQueryResult := sRes; // OUTPUT

METH_ComposeProcessOutboundBox := iRes;
                        
END_METHOD
END_PROGRAM

PROGRAM prgDBQuerierLogger
  VAR
    xTB_GetMissionID : BOOL;  (* generic variables *)
    xIsSQLQueryAllowed : BOOL;
    pInterpDest : __XWORD;
    uiDimInterpDest : UINT;
    xIsValidRef_SQLQueryReq : BOOL;
    pTmp : __XWORD;
    itfInterpreter : SysD_DB.ITF_DBQueryInterpret;
    xTB_InsertLogEntry : BOOL;
    xNewRowSuccessfullyInserted : BOOL;
    xTB_GetLogEntry : BOOL;
    xIsValidRequestedAction : BOOL;
    diActionID : DINT;
    LogEntry : SysD_log_entry_t;  (* eWantedRequestedAction: SAPA_type_of_request_enum_t; sContainerCategory: SysD_Geek.SysD_Geek_container_category_t; *)
    diQueryLength : DINT;
    eQueryError : SysD_DB.ERROR;
    xMessages : BOOL := TRUE;  (* --------------------- filters *)
    xWarnings : BOOL := TRUE;
    xErrors : BOOL := TRUE;
    xFilterByDate : BOOL;
    sFilter_LastEventDT : STRING;
    xFilterByComponent : BOOL;
    sFilter_Component : STRING;
    xContinueGetLog : BOOL;
    sAux : STRING(255);  (* --------------------- *)
    udiEntriesToInsert : UDINT;
    itfElement : COL.IElement;
    ePollRes : COL.COLLECTION_ERROR;
    xResult : BOOL;
    LogEntryToInsert : SysD_log_entry_t;
    xLogEntryIsValid : BOOL;
    xTb_TestInsertNewEntry : BOOL;
    LogEntryTest : SysD_log_entry_t := (sComponent := 'TESTER', sDescription := 'test entry');
    eAddRes : COL.COLLECTION_ERROR;
    eLogEntryFactErr : FBF.ERROR;
    diCounter : DINT;
    xFullBuffer : BOOL;
    diLastNonNullLogID : DINT;
    udiDimExtendedLog : UDINT;
    udiDimLog : UDINT;
    udiLastNonNullArrInd : UDINT;
    xIsEmptyArray : BOOL;
    xAppendToExtendedLog : BOOL;
    xExtendedLogIsFull : BOOL;
    xTB_ContinueLog : BOOL;
    xIsInsertFailed : BOOL;
    xTB_GetLog : BOOL;
    xInit : BOOL := TRUE;
    FB_QuerySQL_0 : SysD_DB.FB_QuerySQL;  (* GENERIC QUERYSQL *)
    CTRL_Query : SysD_DB.SysD_DB_querier_ctrl_struct_t;
    eMySQLAction : SysD_DB.SysD_DB_actions_enum_t;
    REF_REQ_SQLQuery : REFERENCE TO SysDesignBasic.FB_SysD_RequestDetail;
    REF_REQ_Dummy : SysDesignBasic.FB_SysD_RequestDetail;
    iCountSuccess : INT;  (* counters *)
    iCountFailure : INT;
    eLastQuerierError : SysD_DB.ERROR_QUERIER;  (* errors *)
    eLastInterpError : SysD_DB.ERROR;
    eLastSysD_DB_Error : SysD_DB.ERROR;
    eLastMySQLError : SysD_DB.MySQL.ERROR;
    pDB_INQueue : POINTER TO COL.Queue;  (* pointers to collection elements *)
    pDB_OUTHashTable : POINTER TO COL.IMap;
    asIN_LogEntries : ARRAY[0..49] OF ILogEntry;  (* QUEUE IN *)
    itfQueue_LogEntries : COL.Queue := (paElements := ADR(asIN_LogEntries), udiMaxElements := ANY_TO_UDINT((XSIZEOF(asIN_LogEntries) / XSIZEOF(asIN_LogEntries[0]))));
    itfLogEntryElement : ILogEntry;
    LogEntriesFactory : LogEntryElementFactory;
    xMultiInsertMode : BOOL := TRUE;
    sQuery : SysD_DB.SysD_MySQLQuery;  (* get mission ID *)
    asMySQLCommand : SysD_DB.SysD_MySQLCommand;
    diGMSInstanceID : DINT := 100;  (* SQL_Interp_GetMissionId_0: SQL_Interp_GetMissionId;// interpreters *)
    diAuxMissionID : DINT;
    xIsValidMissionID : BOOL;
    diMissionID : DINT;  (* uiDimMissionIDArr: UINT := 1; *)
    R_TRIG_GetMissionSuccess : R_TRIG;
    R_TRIG_GetMissionFailure : R_TRIG;
    REQ_GetMissionID : SysDesignBasic.FB_SysD_RequestDetail;
  END_VAR
  VAR CONSTANT
    c_uiMultiInsertStringSize : UINT := ANY_TO_UINT(((SysD_DB.MySQL.gc_MySQL_Parameter.gc_MySQL_iStatementMax + 1) * SysD_DB.MySQL.gc_MySQL_Parameter.gc_MySQL_iStatementLength));
  END_VAR
  VAR
    sMultiInsertQuery : STRING(c_uiMultiInsertStringSize);  (* 07/11/2022: multi insert sMultiInsertQuery : SysD_DB.SysD_MySQLQuery; *)
    diMultiInsertQueryLen : DINT;
    sPeekQuery : SysD_DB.SysD_MySQLQuery;
    diPeekQueryLen : DINT;
    xTB_MultiInsertLogEntries : BOOL;
    diSumQueryLen : DINT;
    ePeekRes : COL.COLLECTION_ERROR;
    eRemoveRes : COL.COLLECTION_ERROR;
    xAddToMultiInsert : BOOL;
    diMaxQueryLen : DINT;
    xConcatRes : BOOL;
    REQ_InsertLogEntry : SysDesignBasic.FB_SysD_RequestDetail;  (* insert new action sNewAction_Station: STRING := 'S01'; eNewAction_TypeOfRequest: SAPA_type_of_request_enum_t := SAPA_type_of_request_enum_t.PICK_UP; xNewAction_IsAutomatic: BOOL; *)
    R_TRIG_InsertActionSuccess : Standard.R_TRIG;
    R_TRIG_InsertActionFailure : Standard.R_TRIG;
    REQ_GetLog : SysDesignBasic.FB_SysD_RequestDetail;  (* get new action *)
    SQL_Interp_GetLog_0 : SQL_Interp_GetLog;
    R_TRIG_GetLogSuccess : R_TRIG;
    R_TRIG_GetLogFailure : R_TRIG;
    SysD_DB_Input : SysD_DB.SysD_db_input_struct_t := (sHost := GVL_Constants.gc_sTESTDatabaseIP, sDatabase := GVL_Constants.gc_sTESTDatabaseName, sUsername := 'plc_user', sPassword := 'deb11_mySQL');  (* database specific *)
    aLog : ARRAY[0..39] OF SysD_log_row_t;
    aExtendedLog : ARRAY[0..119] OF SysD_log_row_t;
  END_VAR
  VAR CONSTANT
    c_sCallerName : STRING := 'Logger';  (* IEC program specific *)
  END_VAR

                    pDB_INQueue := ADR(prgDBExecutor.itfINQueue_MySQLRequest);
pDB_OUTHashTable := ADR(prgDBExecutor.itfOUTHashTable_MySQLResult);

udiDimExtendedLog := TO_UDINT(XSIZEOF(aExtendedLog)/XSIZEOF(aExtendedLog[0]));
udiDimLog := TO_UDINT(XSIZEOF(aLog)/XSIZEOF(aLog[0]));

ACT_CheckReferences();
(*====================================================*)
//01/12/2022: set db
// SysD_DB_Input.sHost := GVL.g_sIPCurrentDB; //02/12/2022
// SysD_DB_Input.sDatabase := GVL.g_sNameCurrentDB; //15/03/2023
(*====================================================*)
// insert new request test
IF xTb_TestInsertNewEntry THEN
	xTb_TestInsertNewEntry := FALSE;
	eAddRes := METH_AddEntryToQueue(
		LogEntry := LogEntryTest, 
		pdiCounter := ADR(diCounter),
		xFullBuffer => xFullBuffer
	);
ELSIF xInit (*AND GVL.g_xCurrentDBIsSet*) THEN //14/11/2022
	xInit := FALSE;
// 	SysD_DB_Input.sHost := GVL.g_sIPCurrentDB; //02/12/2022
// 	SysD_DB_Input.sDatabase := GVL.g_sNameCurrentDB; //15/03/2023
	LogEntry.eSeverity := SysD_log_entry_severity_enum_t.Message;
	LogEntry.sComponent := c_sCallerName;
	LogEntry.sDescription := 'PLC STARTED';
	eAddRes := METH_AddEntryToQueue(
		LogEntry := LogEntry, 
		pdiCounter := ADR(diCounter),
		xFullBuffer => xFullBuffer
	);
END_IF

xIsSQLQueryAllowed := NOT CTRL_Query.xExecute; //01/12/2022: aggiungo condizione per fare in modo di sapere che DB sto usando prima della prima entry

udiEntriesToInsert := itfQueue_LogEntries.CountElements();
IF udiEntriesToInsert > 0 AND xIsSQLQueryAllowed THEN
	IF xMultiInsertMode THEN
		ACT_MultiInsert();
	ELSE
		ACT_SingleInsert();
	END_IF
	
END_IF

(*====================================================*)
//02/11/2022: high level commands
IF xTB_ContinueLog THEN //02/11/2022
	xTB_ContinueLog := FALSE;
	xAppendToExtendedLog := TRUE;
	xTB_GetLogEntry := TRUE;
ELSIF xTB_GetLog THEN
	xTB_GetLog := FALSE;
	SysMem.SysMemSet(pDest := ADR(aExtendedLog), udiCount := XSIZEOF(aExtendedLog), udiValue := 0);
	xAppendToExtendedLog := FALSE;
	xTB_GetLogEntry := TRUE;
END_IF
(*====================================================*)
IF xIsSQLQueryAllowed THEN
	IF xTB_InsertLogEntry THEN // exec
		xTB_InsertLogEntry := FALSE;
		SysMem.SysMemSet(pDest := ADR(asMySQLCommand), udiCount := XSIZEOF(asMySQLCommand), udiValue := 0);
		CTRL_Query.xExecute := TRUE;
		ACT_InsertLogEntry_Request();
		REF_REQ_SQLQuery.METH_SetRequested();
	ELSIF xTB_MultiInsertLogEntries THEN //07/11/2022
		xTB_MultiInsertLogEntries := FALSE;
		SysMem.SysMemSet(pDest := ADR(asMySQLCommand), udiCount := XSIZEOF(asMySQLCommand), udiValue := 0);
		CTRL_Query.xExecute := TRUE;
		ACT_MultiInsertLogEntry_Request();
		REF_REQ_SQLQuery.METH_SetRequested();
	ELSIF xTB_GetLogEntry THEN // query
		xTB_GetLogEntry := FALSE;
		SysMem.SysMemSet(pDest := ADR(asMySQLCommand), udiCount := XSIZEOF(asMySQLCommand), udiValue := 0);
		CTRL_Query.xExecute := TRUE;
		ACT_GetLog_Request();
		REF_REQ_SQLQuery.METH_SetRequested();
	END_IF
END_IF
(*---------------------------------------------------------------*)
ACT_SQLQuery();
(*---------------------------------------------------------------*)
// insert new action request
R_TRIG_InsertActionSuccess(CLK := REQ_InsertLogEntry.METH_IsSuccess());
IF R_TRIG_InsertActionSuccess.Q THEN
	ACT_InsertLogEntry_Success();
END_IF

R_TRIG_InsertActionFailure(CLK := REQ_InsertLogEntry.METH_IsFailure());
IF R_TRIG_InsertActionFailure.Q THEN
	ACT_InsertLogEntry_Failure();
END_IF

pTmp := ADR(xNewRowSuccessfullyInserted); //debug
(*---------------------------------------------------------------*)
// get requested actions
xIsValidRequestedAction := REQ_GetLog.METH_IsSuccess();

R_TRIG_GetLogSuccess(CLK := REQ_GetLog.METH_IsSuccess());
IF R_TRIG_GetLogSuccess.Q THEN
	ACT_GetLog_Success();
	xAppendToExtendedLog := FALSE; //02/11/2022
END_IF

R_TRIG_GetLogFailure(CLK := REQ_GetLog.METH_IsFailure());
IF R_TRIG_GetLogFailure.Q THEN
	ACT_GetLog_Failure();
	xAppendToExtendedLog := FALSE; //02/11/2022
END_IF

pTmp := ADR(aLog[0].sComponent); //debug
(*---------------------------------------------------------------*)
// extended log
diLastNonNullLogID := METH_GetLastNonNullID(
	pLog := ADR(aExtendedLog), udiDim := udiDimExtendedLog,
	udiArrayInd => udiLastNonNullArrInd,
	xEmptyArray => xIsEmptyArray
);
xExtendedLogIsFull := udiLastNonNullArrInd = (udiDimExtendedLog-1);
                  

ACTION ACT_SQLQuery:
                        FB_QuerySQL_0(
	xExecute := CTRL_Query.xExecute, //CBML
	xAbort := CTRL_Query.xAbort, //CBML
	
	xBusy => CTRL_Query.xProcessing, //CBML
	
	xDone => CTRL_Query.xSuccess, //CBML
	xError => CTRL_Query.xFailure, //CBML
	xAborted => CTRL_Query.xAborted, //CBML
	
	eErrorID => CTRL_Query.eErrorQuerier, // error
	eInterpError => CTRL_Query.eInterpError, // error
	eSysD_DB_Error => CTRL_Query.eSysD_DB_Error, // error
	eMySQLError => CTRL_Query.eMySQLError, // error
	udiAffetedRows => CTRL_Query.udiAffectedRows, // 28/06/2022: affected rows
	
	sCaller := c_sCallerName, // caller name shoud be unique per IEC program
	
	SysD_DB_Input := SysD_DB_Input, // database parameters
	asMySQLCommand := asMySQLCommand, // specific for what we're looking for
	
	eMySQLAction := eMySQLAction, //28/06/2022: expansion to exec
	pDest := pInterpDest, // specific for what we're looking for
	uiDim := uiDimInterpDest, // specific for what we're looking for
	itfInterpreter := itfInterpreter, // specific for what we're looking for
	
	pDB_INQueue := pDB_INQueue, // queue of sql requests
	pDB_OUTHashTable := pDB_OUTHashTable // hashtable of sql results
);
CTRL_Query.xTerminated := CTRL_Query.xSuccess OR CTRL_Query.xFailure OR CTRL_Query.xAborted;
IF CTRL_Query.xTerminated THEN
	// saving last errors
	eLastQuerierError := CTRL_Query.eErrorQuerier;
	eLastInterpError := CTRL_Query.eInterpError;
	eLastSysD_DB_Error := CTRL_Query.eSysD_DB_Error;
	eLastMySQLError := CTRL_Query.eMySQLError;
	
	// result-specific stuff to always do
	IF CTRL_Query.xSuccess THEN
		iCountSuccess := (iCountSuccess + 1) MOD 16#7FFF;
		REF_REQ_SQLQuery.METH_SetSuccess();
	ELSE
		REF_REQ_SQLQuery.METH_SetFailure();
		iCountFailure := (iCountFailure + 1) MOD 16#7FFF;
		IF CTRL_Query.xAborted THEN
			//
		ELSIF CTRL_Query.xFailure THEN
			//
		END_IF 
	END_IF
	CTRL_Query.xExecute := FALSE;
	FB_QuerySQL_0(xExecute := FALSE);
END_IF

                      
END_ACTION

ACTION ACT_CheckReferences:
                        xIsValidRef_SQLQueryReq := __ISVALIDREF(REF_REQ_SQLQuery);
IF NOT xIsValidRef_SQLQueryReq THEN
	REF_REQ_SQLQuery REF= REF_REQ_Dummy;
END_IF
                      
END_ACTION

ACTION ACT_InsertLogEntry_Request:
                        sQuery := '';
sQuery := FUN_DB_insert_log_entry(
	SysD_LogEntry := LogEntryToInsert,
);

diQueryLength := STU.StrLenA(pstData := ADR(sQuery));

eQueryError := SysD_DB.FUN_Query2SQLCmd(
	pbQuery := ADR(sQuery), 
	asSQLCommand => asMySQLCommand,
	diQueryLength := diQueryLength,
);

pInterpDest := 0;
uiDimInterpDest := 0;

itfInterpreter := 0;

REF_REQ_SQLQuery REF= REQ_InsertLogEntry;

eMySQLAction := SysD_DB.SysD_DB_actions_enum_t.Exec;

xNewRowSuccessfullyInserted := FALSE;
                      
END_ACTION

ACTION ACT_InsertLogEntry_Failure:
                        IF CTRL_Query.xAborted THEN
	//
ELSIF CTRL_Query.xFailure THEN
	//
END_IF

                      
END_ACTION

ACTION ACT_InsertLogEntry_Success:
                        xNewRowSuccessfullyInserted := FALSE;
IF CTRL_Query.udiAffectedRows > 0 THEN
	xNewRowSuccessfullyInserted := TRUE;
END_IF
                      
END_ACTION

ACTION ACT_MultiInsertLogEntry_Request:
                        // sQuery := '';
// sQuery := FUN_DB_insert_log_entry(
// 	SysD_LogEntry := LogEntryToInsert,
// );
// 
// diQueryLength := STU.StrLenA(pstData := ADR(sQuery));

// 07/11/2022: QUERY IS COMPOSED ELSEWHERE!!!
// sQuery := sMultiInsertQuery;
diQueryLength := STU.StrLenA(pstData := ADR(sMultiInsertQuery));

eQueryError := SysD_DB.FUN_Query2SQLCmd(
	pbQuery := ADR(sMultiInsertQuery), 
	asSQLCommand => asMySQLCommand,
	diQueryLength := diQueryLength,
);

pInterpDest := 0;
uiDimInterpDest := 0;

itfInterpreter := 0;

REF_REQ_SQLQuery REF= REQ_InsertLogEntry;

eMySQLAction := SysD_DB.SysD_DB_actions_enum_t.Exec;

xNewRowSuccessfullyInserted := FALSE;
                      
END_ACTION

ACTION ACT_GetLog_Failure:
                        IF CTRL_Query.xAborted THEN
	//
ELSIF CTRL_Query.xFailure THEN
	//
END_IF

                      
END_ACTION

ACTION ACT_GetLog_Request:
                        	
sQuery := '';
IF xMessages AND xWarnings AND xErrors THEN
	sQuery := 'select * from t_log where (severity = 0 OR severity = 1 OR severity = 2)';
	
ELSIF NOT xMessages AND xWarnings AND xErrors THEN
	sQuery := 'select * from t_log where (severity = 1 OR severity = 2)';
ELSIF xMessages AND NOT xWarnings AND xErrors THEN
	sQuery := 'select * from t_log where (severity = 0 OR severity = 2)';
ELSIF xMessages AND xWarnings AND NOT xErrors THEN
	sQuery := 'select * from t_log where (severity = 0 OR severity = 1)';

ELSIF xMessages AND NOT xWarnings AND NOT xErrors THEN
	sQuery := 'select * from t_log where severity = 0';
ELSIF NOT xMessages AND xWarnings AND NOT xErrors THEN
	sQuery := 'select * from t_log where severity = 1';
ELSIF NOT xMessages AND NOT xWarnings AND xErrors THEN
	sQuery := 'select * from t_log where severity = 2';
	
